  MoveL 4740 to (-40.39, 151.7, 78.65) mm, rotated rx -180 ry 0 rz 180 deg; joints [-52.89, -15.203, 87.582, 77.101, 54.898, -68.284]
  MoveL 4741 to (-40.39, 151.7, 78.65) mm, rotated rx -180 ry 0 rz 180 deg; joints [-52.89, -15.203, 87.582, 77.101, 54.898, -68.284]
  Call Extruder(10.98377)
  MoveL 4742 to (-40.44, 151.45, 78.65) mm, rotated rx 180 ry 0 rz -180 deg; joints [-52.871, -15.235, 87.606, 77.086, 54.882, -68.269]
  MoveL 4743 to (-40.44, 151.45, 78.65) mm, rotated rx 180 ry 0 rz -180 deg; joints [-52.871, -15.235, 87.606, 77.086, 54.882, -68.269]
  Call Extruder(11.11830)
  MoveL 4744 to (-40.49, 151.2, 78.65) mm, rotated rx 180 ry 0 rz 180 deg; joints [-52.853, -15.267, 87.629, 77.072, 54.867, -68.254]
  MoveL 4745 to (-40.49, 151.2, 78.65) mm, rotated rx 180 ry 0 rz 180 deg; joints [-52.853, -15.267, 87.629, 77.072, 54.867, -68.254]
  Call Extruder(11.25223)
  MoveL 4746 to (-40.54, 150.95, 78.65) mm, rotated rx 180 ry 0 rz 180 deg; joints [-52.834, -15.299, 87.653, 77.057, 54.851, -68.239]
  MoveL 4747 to (-40.54, 150.95, 78.65) mm, rotated rx 180 ry 0 rz 180 deg; joints [-52.834, -15.299, 87.653, 77.057, 54.851, -68.239]
  Call Extruder(11.40008)
  MoveL 4748 to (-40.59, 150.67, 78.65) mm, rotated rx 180 ry 0 rz 180 deg; joints [-52.812, -15.334, 87.679, 77.041, 54.833, -68.222]
  MoveL 4749 to (-40.59, 150.67, 78.65) mm, rotated rx 180 ry 0 rz 180 deg; joints [-52.812, -15.334, 87.679, 77.041, 54.833, -68.222]
  Call Extruder(11.56181)
  MoveL 4750 to (-40.64, 150.37, 78.65) mm, rotated rx -180 ry 0 rz -180 deg; joints [-52.787, -15.372, 87.707, 77.023, 54.812, -68.203]
  MoveL 4751 to (-40.64, 150.37, 78.65) mm, rotated rx -180 ry 0 rz -180 deg; joints [-52.787, -15.372, 87.707, 77.023, 54.812, -68.203]
  Call Extruder(11.72281)
  MoveL 4752 to (-40.69, 150.06, 78.65) mm, rotated rx -180 ry 0 rz 180 deg; joints [-52.762, -15.411, 87.735, 77.004, 54.791, -68.184]
  MoveL 4753 to (-40.69, 150.06, 78.65) mm, rotated rx -180 ry 0 rz 180 deg; joints [-52.762, -15.411, 87.735, 77.004, 54.791, -68.184]
  Call Extruder(11.88308)
  MoveL 4754 to (-40.74, 149.76, 78.65) mm, rotated rx 180 ry 0 rz 180 deg; joints [-52.737, -15.449, 87.762, 76.986, 54.771, -68.165]
  MoveL 4755 to (-40.74, 149.76, 78.65) mm, rotated rx 180 ry 0 rz 180 deg; joints [-52.737, -15.449, 87.762, 76.986, 54.771, -68.165]
  Call Extruder(12.04262)
  MoveL 4756 to (-40.78, 149.45, 78.65) mm, rotated rx 180 ry 0 rz 180 deg; joints [-52.712, -15.487, 87.79, 76.967, 54.75, -68.146]
  MoveL 4757 to (-40.78, 149.45, 78.65) mm, rotated rx 180 ry 0 rz 180 deg; joints [-52.712, -15.487, 87.79, 76.967, 54.75, -68.146]
  Call Extruder(12.20143)
  MoveL 4758 to (-40.83, 149.14, 78.65) mm, rotated rx -180 ry 0 rz -180 deg; joints [-52.687, -15.526, 87.818, 76.949, 54.729, -68.127]
  MoveL 4759 to (-40.83, 149.14, 78.65) mm, rotated rx -180 ry 0 rz -180 deg; joints [-52.687, -15.526, 87.818, 76.949, 54.729, -68.127]
  Call Extruder(12.38010)
  MoveL 4760 to (-40.88, 148.8, 78.65) mm, rotated rx 180 ry 0 rz 180 deg; joints [-52.658, -15.568, 87.849, 76.927, 54.704, -68.106]
  MoveL 4761 to (-40.88, 148.8, 78.65) mm, rotated rx 180 ry 0 rz 180 deg; joints [-52.658, -15.568, 87.849, 76.927, 54.704, -68.106]
  Call Extruder(12.57854)
  MoveL 4762 to (-40.92, 148.41, 78.65) mm, rotated rx 180 ry 0 rz 180 deg; joints [-52.624, -15.615, 87.883, 76.903, 54.675, -68.081]
  MoveL 4763 to (-40.92, 148.41, 78.65) mm, rotated rx 180 ry 0 rz 180 deg; joints [-52.624, -15.615, 87.883, 76.903, 54.675, -68.081]
  Call Extruder(12.77611)
  MoveL 4764 to (-40.97, 148.02, 78.65) mm, rotated rx 180 ry 0 rz -180 deg; joints [-52.59, -15.662, 87.917, 76.878, 54.647, -68.057]
  MoveL 4765 to (-40.97, 148.02, 78.65) mm, rotated rx 180 ry 0 rz -180 deg; joints [-52.59, -15.662, 87.917, 76.878, 54.647, -68.057]
  Call Extruder(12.97282)
  MoveL 4766 to (-41.02, 147.63, 78.65) mm, rotated rx -180 ry 0 rz 180 deg; joints [-52.556, -15.709, 87.951, 76.854, 54.618, -68.032]
  MoveL 4767 to (-41.02, 147.63, 78.65) mm, rotated rx -180 ry 0 rz 180 deg; joints [-52.556, -15.709, 87.951, 76.854, 54.618, -68.032]
  Call Extruder(13.16866)
  MoveL 4768 to (-41.06, 147.25, 78.65) mm, rotated rx 180 ry 0 rz 180 deg; joints [-52.521, -15.756, 87.985, 76.829, 54.589, -68.008]
  MoveL 4769 to (-41.06, 147.25, 78.65) mm, rotated rx 180 ry 0 rz 180 deg; joints [-52.521, -15.756, 87.985, 76.829, 54.589, -68.008]
  Call Extruder(13.46406)
  MoveL 4770 to (-41.11, 146.66, 78.65) mm, rotated rx -180 ry 0 rz 180 deg; joints [-52.466, -15.826, 88.036, 76.79, 54.543, -67.97]
  MoveL 4771 to (-41.11, 146.66, 78.65) mm, rotated rx -180 ry 0 rz 180 deg; joints [-52.466, -15.826, 88.036, 76.79, 54.543, -67.97]
  Call Extruder(13.75812)
  MoveL 4772 to (-41.15, 146.07, 78.65) mm, rotated rx 180 ry 0 rz 180 deg; joints [-52.411, -15.895, 88.086, 76.751, 54.496, -67.932]
  MoveL 4773 to (-41.15, 146.07, 78.65) mm, rotated rx 180 ry 0 rz 180 deg; joints [-52.411, -15.895, 88.086, 76.751, 54.496, -67.932]
  Call Extruder(14.05086)
  MoveL 4774 to (-41.2, 145.48, 78.65) mm, rotated rx -180 ry 0 rz 180 deg; joints [-52.355, -15.964, 88.136, 76.712, 54.449, -67.894]
  MoveL 4775 to (-41.2, 145.48, 78.65) mm, rotated rx -180 ry 0 rz 180 deg; joints [-52.355, -15.964, 88.136, 76.712, 54.449, -67.894]
  Call Extruder(14.62431)
  MoveL 4776 to (-41.25, 144.32, 78.65) mm, rotated rx -180 ry 0 rz 180 deg; joints [-52.239, -16.097, 88.231, 76.632, 54.349, -67.818]
  MoveL 4777 to (-41.25, 144.32, 78.65) mm, rotated rx -180 ry 0 rz 180 deg; joints [-52.239, -16.097, 88.231, 76.632, 54.349, -67.818]
  Call Extruder(15.33827)
  MoveL 4778 to (-41.29, 142.86, 78.65) mm, rotated rx 180 ry 0 rz 180 deg; joints [-52.09, -16.261, 88.348, 76.53, 54.222, -67.722]
  Call Extruder(57.40309)
  MoveL 4779 to (-41.29, 57.14, 78.65) mm, rotated rx 180 ry 0 rz 180 deg; joints [-40.759, -24.748, 93.754, 67.429, 44.994, -59.555]
  Call Extruder(57.83164)
  MoveL 4780 to (-41.27, 56.26, 78.65) mm, rotated rx 180 ry 0 rz 180 deg; joints [-40.614, -24.821, 93.795, 67.296, 44.882, -59.439]
  MoveL 4781 to (-41.27, 56.26, 78.65) mm, rotated rx 180 ry 0 rz 180 deg; joints [-40.614, -24.821, 93.795, 67.296, 44.882, -59.439]
  Call Extruder(58.40509)
  MoveL 4782 to (-41.22, 55.1, 78.65) mm, rotated rx -180 ry 0 rz 180 deg; joints [-40.419, -24.917, 93.848, 67.115, 44.73, -59.283]
  MoveL 4783 to (-41.22, 55.1, 78.65) mm, rotated rx -180 ry 0 rz 180 deg; joints [-40.419, -24.917, 93.848, 67.115, 44.73, -59.283]
  Call Extruder(58.83941)
  MoveL 4784 to (-41.18, 54.23, 78.65) mm, rotated rx 180 ry 0 rz 180 deg; joints [-40.269, -24.987, 93.887, 66.976, 44.613, -59.164]
  MoveL 4785 to (-41.18, 54.23, 78.65) mm, rotated rx 180 ry 0 rz 180 deg; joints [-40.269, -24.987, 93.887, 66.976, 44.613, -59.164]
  Call Extruder(59.13347)
  MoveL 4786 to (-41.13, 53.64, 78.65) mm, rotated rx 180 ry 0 rz -180 deg; joints [-40.165, -25.033, 93.912, 66.882, 44.532, -59.084]
  MoveL 4787 to (-41.13, 53.64, 78.65) mm, rotated rx 180 ry 0 rz -180 deg; joints [-40.165, -25.033, 93.912, 66.882, 44.532, -59.084]
  Call Extruder(59.42887)
  MoveL 4788 to (-41.09, 53.05, 78.65) mm, rotated rx -180 ry 0 rz 180 deg; joints [-40.062, -25.078, 93.937, 66.787, 44.452, -59.003]
  MoveL 4789 to (-41.09, 53.05, 78.65) mm, rotated rx -180 ry 0 rz 180 deg; joints [-40.062, -25.078, 93.937, 66.787, 44.452, -59.003]
  Call Extruder(59.67511)
  MoveL 4790 to (-41.04, 52.56, 78.65) mm, rotated rx -180 ry 0 rz 180 deg; joints [-39.975, -25.115, 93.958, 66.707, 44.384, -58.935]
  MoveL 4791 to (-41.04, 52.56, 78.65) mm, rotated rx -180 ry 0 rz 180 deg; joints [-39.975, -25.115, 93.958, 66.707, 44.384, -58.935]
  Call Extruder(59.87182)
  MoveL 4792 to (-40.99, 52.17, 78.65) mm, rotated rx 180 ry 0 rz 180 deg; joints [-39.904, -25.143, 93.973, 66.643, 44.328, -58.881]
  MoveL 4793 to (-40.99, 52.17, 78.65) mm, rotated rx 180 ry 0 rz 180 deg; joints [-39.904, -25.143, 93.973, 66.643, 44.328, -58.881]
  Call Extruder(60.06939)
  MoveL 4794 to (-40.95, 51.78, 78.65) mm, rotated rx -180 ry 0 rz -180 deg; joints [-39.833, -25.171, 93.989, 66.579, 44.273, -58.827]
  MoveL 4795 to (-40.95, 51.78, 78.65) mm, rotated rx -180 ry 0 rz -180 deg; joints [-39.833, -25.171, 93.989, 66.579, 44.273, -58.827]
  Call Extruder(60.26783)
  MoveL 4796 to (-40.9, 51.4, 78.65) mm, rotated rx 180 ry 0 rz 180 deg; joints [-39.763, -25.199, 94.004, 66.514, 44.217, -58.773]
  MoveL 4797 to (-40.9, 51.4, 78.65) mm, rotated rx 180 ry 0 rz 180 deg; joints [-39.763, -25.199, 94.004, 66.514, 44.217, -58.773]
  Call Extruder(60.46714)
  MoveL 4798 to (-40.86, 51.01, 78.65) mm, rotated rx 180 ry 0 rz 180 deg; joints [-39.692, -25.227, 94.02, 66.45, 44.162, -58.718]
  MoveL 4799 to (-40.86, 51.01, 78.65) mm, rotated rx 180 ry 0 rz 180 deg; joints [-39.692, -25.227, 94.02, 66.45, 44.162, -58.718]
  Call Extruder(60.62596)
  MoveL 4800 to (-40.81, 50.7, 78.65) mm, rotated rx 180 ry 0 rz 180 deg; joints [-39.634, -25.248, 94.031, 66.398, 44.116, -58.675]
  MoveL 4801 to (-40.81, 50.7, 78.65) mm, rotated rx 180 ry 0 rz 180 deg; joints [-39.634, -25.248, 94.031, 66.398, 44.116, -58.675]
  Call Extruder(60.78550)
  MoveL 4802 to (-40.76, 50.4, 78.65) mm, rotated rx 180 ry 0 rz 180 deg; joints [-39.576, -25.269, 94.043, 66.346, 44.07, -58.632]
  MoveL 4803 to (-40.76, 50.4, 78.65) mm, rotated rx 180 ry 0 rz 180 deg; joints [-39.576, -25.269, 94.043, 66.346, 44.07, -58.632]
  Call Extruder(60.94577)
  MoveL 4804 to (-40.71, 50.09, 78.65) mm, rotated rx -180 ry 0 rz 180 deg; joints [-39.518, -25.29, 94.054, 66.294, 44.025, -58.588]
  MoveL 4805 to (-40.71, 50.09, 78.65) mm, rotated rx -180 ry 0 rz 180 deg; joints [-39.518, -25.29, 94.054, 66.294, 44.025, -58.588]
  Call Extruder(61.10677)
  MoveL 4806 to (-40.66, 49.79, 78.65) mm, rotated rx -180 ry 0 rz 180 deg; joints [-39.46, -25.31, 94.065, 66.241, 43.979, -58.545]
  MoveL 4807 to (-40.66, 49.79, 78.65) mm, rotated rx -180 ry 0 rz 180 deg; joints [-39.46, -25.31, 94.065, 66.241, 43.979, -58.545]
  Call Extruder(61.26850)
  MoveL 4808 to (-40.61, 49.48, 78.65) mm, rotated rx 180 ry 0 rz 180 deg; joints [-39.402, -25.331, 94.077, 66.189, 43.933, -58.501]
  MoveL 4809 to (-40.61, 49.48, 78.65) mm, rotated rx 180 ry 0 rz 180 deg; joints [-39.402, -25.331, 94.077, 66.189, 43.933, -58.501]
  Call Extruder(61.43095)
  MoveL 4810 to (-40.57, 49.17, 78.65) mm, rotated rx 180 ry 0 rz 180 deg; joints [-39.344, -25.352, 94.088, 66.136, 43.888, -58.457]
  MoveL 4811 to (-40.57, 49.17, 78.65) mm, rotated rx 180 ry 0 rz 180 deg; joints [-39.344, -25.352, 94.088, 66.136, 43.888, -58.457]
  Call Extruder(61.56487)
  MoveL 4812 to (-40.52, 48.92, 78.65) mm, rotated rx -180 ry 0 rz 180 deg; joints [-39.296, -25.368, 94.096, 66.092, 43.849, -58.421]
  MoveL 4813 to (-40.52, 48.92, 78.65) mm, rotated rx -180 ry 0 rz 180 deg; joints [-39.296, -25.368, 94.096, 66.092, 43.849, -58.421]
  Call Extruder(61.69941)
  MoveL 4814 to (-40.47, 48.68, 78.65) mm, rotated rx 180 ry 0 rz 180 deg; joints [-39.247, -25.383, 94.105, 66.049, 43.81, -58.385]
  MoveL 4815 to (-40.47, 48.68, 78.65) mm, rotated rx 180 ry 0 rz 180 deg; joints [-39.247, -25.383, 94.105, 66.049, 43.81, -58.385]
  Call Extruder(61.83455)
  MoveL 4816 to (-40.42, 48.43, 78.65) mm, rotated rx 180 ry 0 rz 180 deg; joints [-39.198, -25.399, 94.114, 66.005, 43.772, -58.349]
  MoveL 4817 to (-40.42, 48.43, 78.65) mm, rotated rx 180 ry 0 rz 180 deg; joints [-39.198, -25.399, 94.114, 66.005, 43.772, -58.349]
  Call Extruder(61.97031)
  MoveL 4818 to (-40.37, 48.18, 78.65) mm, rotated rx 180 ry 0 rz 180 deg; joints [-39.149, -25.415, 94.122, 65.961, 43.733, -58.313]
  MoveL 4819 to (-40.37, 48.18, 78.65) mm, rotated rx 180 ry 0 rz 180 deg; joints [-39.149, -25.415, 94.122, 65.961, 43.733, -58.313]
  Call Extruder(62.10667)
  MoveL 4820 to (-40.32, 47.93, 78.65) mm, rotated rx -180 ry 0 rz 180 deg; joints [-39.1, -25.43, 94.131, 65.917, 43.694, -58.276]
  MoveL 4821 to (-40.32, 47.93, 78.65) mm, rotated rx -180 ry 0 rz 180 deg; joints [-39.1, -25.43, 94.131, 65.917, 43.694, -58.276]
  Call Extruder(62.24365)
  MoveL 4822 to (-40.27, 47.68, 78.65) mm, rotated rx 180 ry 0 rz 180 deg; joints [-39.051, -25.446, 94.139, 65.873, 43.656, -58.24]
  MoveL 4823 to (-40.27, 47.68, 78.65) mm, rotated rx 180 ry 0 rz 180 deg; joints [-39.051, -25.446, 94.139, 65.873, 43.656, -58.24]
  Call Extruder(62.38124)
  MoveL 4824 to (-40.22, 47.43, 78.65) mm, rotated rx -180 ry 0 rz 180 deg; joints [-39.002, -25.461, 94.148, 65.829, 43.617, -58.204]
  MoveL 4825 to (-40.22, 47.43, 78.65) mm, rotated rx -180 ry 0 rz 180 deg; joints [-39.002, -25.461, 94.148, 65.829, 43.617, -58.204]
  Call Extruder(62.49496)
  MoveL 4826 to (-40.17, 47.23, 78.65) mm, rotated rx 180 ry 0 rz 180 deg; joints [-38.962, -25.474, 94.154, 65.792, 43.585, -58.174]
  MoveL 4827 to (-40.17, 47.23, 78.65) mm, rotated rx 180 ry 0 rz 180 deg; joints [-38.962, -25.474, 94.154, 65.792, 43.585, -58.174]
  Call Extruder(62.60914)
  MoveL 4828 to (-40.13, 47.02, 78.65) mm, rotated rx -180 ry 0 rz 180 deg; joints [-38.921, -25.486, 94.161, 65.755, 43.552, -58.143]
  MoveL 4829 to (-40.13, 47.02, 78.65) mm, rotated rx -180 ry 0 rz 180 deg; joints [-38.921, -25.486, 94.161, 65.755, 43.552, -58.143]
  Call Extruder(62.72378)
  MoveL 4830 to (-40.08, 46.82, 78.65) mm, rotated rx -180 ry 0 rz 180 deg; joints [-38.88, -25.498, 94.168, 65.719, 43.52, -58.113]
  MoveL 4831 to (-40.08, 46.82, 78.65) mm, rotated rx -180 ry 0 rz 180 deg; joints [-38.88, -25.498, 94.168, 65.719, 43.52, -58.113]
  Call Extruder(62.83886)
  MoveL 4832 to (-40.04, 46.61, 78.65) mm, rotated rx 180 ry 0 rz 180 deg; joints [-38.839, -25.511, 94.175, 65.682, 43.488, -58.083]
  MoveL 4833 to (-40.04, 46.61, 78.65) mm, rotated rx 180 ry 0 rz 180 deg; joints [-38.839, -25.511, 94.175, 65.682, 43.488, -58.083]
  Call Extruder(62.96110)
  MoveL 4834 to (-39.98, 46.4, 78.65) mm, rotated rx 180 ry 0 rz -180 deg; joints [-38.795, -25.523, 94.181, 65.643, 43.452, -58.051]
  MoveL 4835 to (-39.98, 46.4, 78.65) mm, rotated rx 180 ry 0 rz -180 deg; joints [-38.795, -25.523, 94.181, 65.643, 43.452, -58.051]
  Call Extruder(63.09076)
  MoveL 4836 to (-39.92, 46.18, 78.65) mm, rotated rx 180 ry 0 rz 180 deg; joints [-38.748, -25.534, 94.187, 65.601, 43.414, -58.018]
  MoveL 4837 to (-39.92, 46.18, 78.65) mm, rotated rx 180 ry 0 rz 180 deg; joints [-38.748, -25.534, 94.187, 65.601, 43.414, -58.018]
  Call Extruder(63.22099)
  MoveL 4838 to (-39.85, 45.95, 78.65) mm, rotated rx -180 ry 0 rz 180 deg; joints [-38.7, -25.546, 94.193, 65.56, 43.376, -57.984]
  MoveL 4839 to (-39.85, 45.95, 78.65) mm, rotated rx -180 ry 0 rz 180 deg; joints [-38.7, -25.546, 94.193, 65.56, 43.376, -57.984]
  Call Extruder(63.35179)
  MoveL 4840 to (-39.78, 45.73, 78.65) mm, rotated rx -180 ry 0 rz 180 deg; joints [-38.653, -25.557, 94.2, 65.518, 43.338, -57.951]
  MoveL 4841 to (-39.78, 45.73, 78.65) mm, rotated rx -180 ry 0 rz 180 deg; joints [-38.653, -25.557, 94.2, 65.518, 43.338, -57.951]
  Call Extruder(63.48315)
  MoveL 4842 to (-39.71, 45.51, 78.65) mm, rotated rx 180 ry 0 rz 180 deg; joints [-38.605, -25.569, 94.206, 65.476, 43.3, -57.917]
  MoveL 4843 to (-39.71, 45.51, 78.65) mm, rotated rx 180 ry 0 rz 180 deg; joints [-38.605, -25.569, 94.206, 65.476, 43.3, -57.917]
  Call Extruder(63.59505)
  MoveL 4844 to (-39.65, 45.32, 78.65) mm, rotated rx 180 ry 0 rz 180 deg; joints [-38.565, -25.578, 94.211, 65.441, 43.268, -57.889]
  MoveL 4845 to (-39.65, 45.32, 78.65) mm, rotated rx 180 ry 0 rz 180 deg; joints [-38.565, -25.578, 94.211, 65.441, 43.268, -57.889]
  Call Extruder(63.70739)
  MoveL 4846 to (-39.59, 45.13, 78.65) mm, rotated rx 180 ry 0 rz 180 deg; joints [-38.524, -25.587, 94.216, 65.405, 43.235, -57.86]
  MoveL 4847 to (-39.59, 45.13, 78.65) mm, rotated rx 180 ry 0 rz 180 deg; joints [-38.524, -25.587, 94.216, 65.405, 43.235, -57.86]
  Call Extruder(63.82018)
  MoveL 4848 to (-39.53, 44.94, 78.65) mm, rotated rx 180 ry 0 rz 180 deg; joints [-38.483, -25.596, 94.221, 65.37, 43.202, -57.832]
  MoveL 4849 to (-39.53, 44.94, 78.65) mm, rotated rx 180 ry 0 rz 180 deg; joints [-38.483, -25.596, 94.221, 65.37, 43.202, -57.832]
  Call Extruder(63.93342)
  MoveL 4850 to (-39.47, 44.75, 78.65) mm, rotated rx 180 ry 0 rz 180 deg; joints [-38.443, -25.605, 94.226, 65.334, 43.169, -57.803]
  MoveL 4851 to (-39.47, 44.75, 78.65) mm, rotated rx 180 ry 0 rz 180 deg; joints [-38.443, -25.605, 94.226, 65.334, 43.169, -57.803]
  Call Extruder(64.04710)
  MoveL 4852 to (-39.41, 44.56, 78.65) mm, rotated rx 180 ry 0 rz 180 deg; joints [-38.402, -25.614, 94.231, 65.298, 43.137, -57.774]
  MoveL 4853 to (-39.41, 44.56, 78.65) mm, rotated rx 180 ry 0 rz 180 deg; joints [-38.402, -25.614, 94.231, 65.298, 43.137, -57.774]
  Call Extruder(64.22906)
  MoveL 4854 to (-39.29, 44.27, 78.65) mm, rotated rx 180 ry 0 rz 180 deg; joints [-38.335, -25.626, 94.237, 65.241, 43.083, -57.729]
  MoveL 4855 to (-39.29, 44.27, 78.65) mm, rotated rx 180 ry 0 rz 180 deg; joints [-38.335, -25.626, 94.237, 65.241, 43.083, -57.729]
  Call Extruder(64.41178)
  MoveL 4856 to (-39.17, 43.98, 78.65) mm, rotated rx -180 ry 0 rz -180 deg; joints [-38.269, -25.637, 94.243, 65.184, 43.028, -57.684]
  MoveL 4857 to (-39.17, 43.98, 78.65) mm, rotated rx -180 ry 0 rz -180 deg; joints [-38.269, -25.637, 94.243, 65.184, 43.028, -57.684]
  Call Extruder(64.58219)
  MoveL 4858 to (-39.05, 43.71, 78.65) mm, rotated rx 180 ry 0 rz 180 deg; joints [-38.207, -25.647, 94.249, 65.131, 42.978, -57.643]
  MoveL 4859 to (-39.05, 43.71, 78.65) mm, rotated rx 180 ry 0 rz 180 deg; joints [-38.207, -25.647, 94.249, 65.131, 42.978, -57.643]
  Call Extruder(64.74017)
  MoveL 4860 to (-38.94, 43.46, 78.65) mm, rotated rx -180 ry 0 rz -180 deg; joints [-38.149, -25.656, 94.253, 65.081, 42.931, -57.604]
  MoveL 4861 to (-38.94, 43.46, 78.65) mm, rotated rx -180 ry 0 rz -180 deg; joints [-38.149, -25.656, 94.253, 65.081, 42.931, -57.604]
  Call Extruder(64.89876)
  MoveL 4862 to (-38.84, 43.21, 78.65) mm, rotated rx 180 ry 0 rz 180 deg; joints [-38.092, -25.666, 94.258, 65.032, 42.884, -57.565]
  MoveL 4863 to (-38.84, 43.21, 78.65) mm, rotated rx 180 ry 0 rz 180 deg; joints [-38.092, -25.666, 94.258, 65.032, 42.884, -57.565]
  Call Extruder(65.10492)
  MoveL 4864 to (-38.66, 42.91, 78.65) mm, rotated rx 180 ry 0 rz 180 deg; joints [-38.016, -25.672, 94.262, 64.969, 42.821, -57.517]
  MoveL 4865 to (-38.66, 42.91, 78.65) mm, rotated rx 180 ry 0 rz 180 deg; joints [-38.016, -25.672, 94.262, 64.969, 42.821, -57.517]
  Call Extruder(65.31187)
  MoveL 4866 to (-38.49, 42.6, 78.65) mm, rotated rx 180 ry 0 rz 180 deg; joints [-37.939, -25.678, 94.265, 64.906, 42.758, -57.469]
  MoveL 4867 to (-38.49, 42.6, 78.65) mm, rotated rx 180 ry 0 rz 180 deg; joints [-37.939, -25.678, 94.265, 64.906, 42.758, -57.469]
  Call Extruder(65.51959)
  MoveL 4868 to (-38.31, 42.3, 78.65) mm, rotated rx 180 ry 0 rz 180 deg; joints [-37.863, -25.685, 94.269, 64.842, 42.695, -57.42]
  MoveL 4869 to (-38.31, 42.3, 78.65) mm, rotated rx 180 ry 0 rz 180 deg; joints [-37.863, -25.685, 94.269, 64.842, 42.695, -57.42]
  Call Extruder(65.72809)
  MoveL 4870 to (-38.14, 41.99, 78.65) mm, rotated rx 180 ry 0 rz -180 deg; joints [-37.787, -25.691, 94.272, 64.779, 42.632, -57.372]
  MoveL 4871 to (-38.14, 41.99, 78.65) mm, rotated rx 180 ry 0 rz -180 deg; joints [-37.787, -25.691, 94.272, 64.779, 42.632, -57.372]
  Call Extruder(65.90765)
  MoveL 4872 to (-37.96, 41.75, 78.65) mm, rotated rx -180 ry 0 rz 180 deg; joints [-37.72, -25.693, 94.273, 64.725, 42.577, -57.332]
  MoveL 4873 to (-37.96, 41.75, 78.65) mm, rotated rx -180 ry 0 rz 180 deg; joints [-37.72, -25.693, 94.273, 64.725, 42.577, -57.332]
  Call Extruder(66.24108)
  MoveL 4874 to (-37.63, 41.3, 78.65) mm, rotated rx 180 ry 0 rz 180 deg; joints [-37.598, -25.695, 94.274, 64.626, 42.474, -57.259]
  MoveL 4875 to (-37.63, 41.3, 78.65) mm, rotated rx 180 ry 0 rz 180 deg; joints [-37.598, -25.695, 94.274, 64.626, 42.474, -57.259]
  Call Extruder(66.57570)
  MoveL 4876 to (-37.3, 40.85, 78.65) mm, rotated rx 180 ry 0 rz 180 deg; joints [-37.475, -25.697, 94.275, 64.527, 42.371, -57.185]
  Call Extruder(67.40363)
  MoveL 4877 to (-36.39, 39.81, 78.65) mm, rotated rx 180 ry 0 rz 180 deg; joints [-37.173, -25.684, 94.268, 64.289, 42.115, -57.012]
  Call Extruder(68.23154)
  MoveL 4878 to (-35.35, 38.9, 78.65) mm, rotated rx -180 ry 0 rz 180 deg; joints [-36.876, -25.647, 94.249, 64.063, 41.859, -56.855]
  Call Extruder(68.39885)
  MoveL 4879 to (-35.13, 38.73, 78.65) mm, rotated rx -180 ry 0 rz 180 deg; joints [-36.818, -25.636, 94.243, 64.02, 41.808, -56.826]
  MoveL 4880 to (-35.13, 38.73, 78.65) mm, rotated rx -180 ry 0 rz 180 deg; joints [-36.818, -25.636, 94.243, 64.02, 41.808, -56.826]
  Call Extruder(68.73227)
  MoveL 4881 to (-34.68, 38.41, 78.65) mm, rotated rx 180 ry 0 rz -180 deg; joints [-36.701, -25.615, 94.231, 63.934, 41.706, -56.767]
  MoveL 4882 to (-34.68, 38.41, 78.65) mm, rotated rx 180 ry 0 rz -180 deg; joints [-36.701, -25.615, 94.231, 63.934, 41.706, -56.767]
  Call Extruder(69.06451)
  MoveL 4883 to (-34.22, 38.08, 78.65) mm, rotated rx 180 ry 0 rz 180 deg; joints [-36.584, -25.593, 94.219, 63.848, 41.603, -56.709]
  MoveL 4884 to (-34.22, 38.08, 78.65) mm, rotated rx 180 ry 0 rz 180 deg; joints [-36.584, -25.593, 94.219, 63.848, 41.603, -56.709]
  Call Extruder(69.18222)
  MoveL 4885 to (-34.05, 37.98, 78.65) mm, rotated rx 180 ry 0 rz -180 deg; joints [-36.544, -25.582, 94.213, 63.82, 41.568, -56.691]
  MoveL 4886 to (-34.05, 37.98, 78.65) mm, rotated rx 180 ry 0 rz -180 deg; joints [-36.544, -25.582, 94.213, 63.82, 41.568, -56.691]
  Call Extruder(69.38994)
  MoveL 4887 to (-33.75, 37.8, 78.65) mm, rotated rx 180 ry 0 rz 180 deg; joints [-36.474, -25.564, 94.203, 63.77, 41.506, -56.658]
  MoveL 4888 to (-33.75, 37.8, 78.65) mm, rotated rx 180 ry 0 rz 180 deg; joints [-36.474, -25.564, 94.203, 63.77, 41.506, -56.658]
  Call Extruder(69.59688)
  MoveL 4889 to (-33.45, 37.63, 78.65) mm, rotated rx -180 ry 0 rz 180 deg; joints [-36.403, -25.546, 94.193, 63.72, 41.443, -56.626]
  MoveL 4890 to (-33.45, 37.63, 78.65) mm, rotated rx -180 ry 0 rz 180 deg; joints [-36.403, -25.546, 94.193, 63.72, 41.443, -56.626]
  Call Extruder(69.80304)
  MoveL 4891 to (-33.14, 37.45, 78.65) mm, rotated rx 180 ry 0 rz -180 deg; joints [-36.333, -25.527, 94.183, 63.67, 41.381, -56.594]
  MoveL 4892 to (-33.14, 37.45, 78.65) mm, rotated rx 180 ry 0 rz -180 deg; joints [-36.333, -25.527, 94.183, 63.67, 41.381, -56.594]
  Call Extruder(69.98473)
  MoveL 4893 to (-32.86, 37.31, 78.65) mm, rotated rx 180 ry 0 rz 180 deg; joints [-36.272, -25.509, 94.173, 63.628, 41.326, -56.567]
  MoveL 4894 to (-32.86, 37.31, 78.65) mm, rotated rx 180 ry 0 rz 180 deg; joints [-36.272, -25.509, 94.173, 63.628, 41.326, -56.567]
  Call Extruder(70.14273)
  MoveL 4895 to (-32.62, 37.2, 78.65) mm, rotated rx 180 ry 0 rz 180 deg; joints [-36.221, -25.491, 94.164, 63.594, 41.28, -56.546]
  MoveL 4896 to (-32.62, 37.2, 78.65) mm, rotated rx 180 ry 0 rz 180 deg; joints [-36.221, -25.491, 94.164, 63.594, 41.28, -56.546]
  Call Extruder(70.30013)
  MoveL 4897 to (-32.37, 37.1, 78.65) mm, rotated rx 180 ry 0 rz -180 deg; joints [-36.17, -25.472, 94.154, 63.56, 41.234, -56.525]
  MoveL 4898 to (-32.37, 37.1, 78.65) mm, rotated rx 180 ry 0 rz -180 deg; joints [-36.17, -25.472, 94.154, 63.56, 41.234, -56.525]
  Call Extruder(70.48284)
  MoveL 4899 to (-32.08, 36.97, 78.65) mm, rotated rx 180 ry 0 rz 180 deg; joints [-36.112, -25.451, 94.142, 63.521, 41.18, -56.502]
  MoveL 4900 to (-32.08, 36.97, 78.65) mm, rotated rx 180 ry 0 rz 180 deg; joints [-36.112, -25.451, 94.142, 63.521, 41.18, -56.502]
  Call Extruder(70.66479)
  MoveL 4901 to (-31.78, 36.85, 78.65) mm, rotated rx 180 ry 0 rz 180 deg; joints [-36.053, -25.429, 94.13, 63.482, 41.127, -56.478]
  MoveL 4902 to (-31.78, 36.85, 78.65) mm, rotated rx 180 ry 0 rz 180 deg; joints [-36.053, -25.429, 94.13, 63.482, 41.127, -56.478]
  Call Extruder(70.81212)
  MoveL 4903 to (-31.54, 36.76, 78.65) mm, rotated rx 180 ry 0 rz 180 deg; joints [-36.006, -25.41, 94.12, 63.451, 41.084, -56.46]
  MoveL 4904 to (-31.54, 36.76, 78.65) mm, rotated rx 180 ry 0 rz 180 deg; joints [-36.006, -25.41, 94.12, 63.451, 41.084, -56.46]
  Call Extruder(70.92535)
  MoveL 4905 to (-31.35, 36.7, 78.65) mm, rotated rx 180 ry 0 rz 180 deg; joints [-35.971, -25.395, 94.111, 63.429, 41.052, -56.447]
  MoveL 4906 to (-31.35, 36.7, 78.65) mm, rotated rx 180 ry 0 rz 180 deg; joints [-35.971, -25.395, 94.111, 63.429, 41.052, -56.447]
  Call Extruder(71.03815)
  MoveL 4907 to (-31.17, 36.64, 78.65) mm, rotated rx -180 ry 0 rz 180 deg; joints [-35.936, -25.38, 94.103, 63.407, 41.02, -56.435]
  MoveL 4908 to (-31.17, 36.64, 78.65) mm, rotated rx -180 ry 0 rz 180 deg; joints [-35.936, -25.38, 94.103, 63.407, 41.02, -56.435]
  Call Extruder(71.15049)
  MoveL 4909 to (-30.98, 36.58, 78.65) mm, rotated rx -180 ry 0 rz -180 deg; joints [-35.901, -25.364, 94.095, 63.384, 40.988, -56.422]
  MoveL 4910 to (-30.98, 36.58, 78.65) mm, rotated rx -180 ry 0 rz -180 deg; joints [-35.901, -25.364, 94.095, 63.384, 40.988, -56.422]
  Call Extruder(71.26240)
  MoveL 4911 to (-30.79, 36.52, 78.65) mm, rotated rx 180 ry 0 rz 180 deg; joints [-35.867, -25.349, 94.086, 63.362, 40.956, -56.409]
  MoveL 4912 to (-30.79, 36.52, 78.65) mm, rotated rx 180 ry 0 rz 180 deg; joints [-35.867, -25.349, 94.086, 63.362, 40.956, -56.409]
  Call Extruder(71.38380)
  MoveL 4913 to (-30.58, 36.45, 78.65) mm, rotated rx -180 ry 0 rz 180 deg; joints [-35.829, -25.332, 94.077, 63.338, 40.921, -56.396]
  MoveL 4914 to (-30.58, 36.45, 78.65) mm, rotated rx -180 ry 0 rz 180 deg; joints [-35.829, -25.332, 94.077, 63.338, 40.921, -56.396]
  Call Extruder(71.51459)
  MoveL 4915 to (-30.36, 36.39, 78.65) mm, rotated rx 180 ry 0 rz 180 deg; joints [-35.788, -25.313, 94.067, 63.313, 40.883, -56.382]
  MoveL 4916 to (-30.36, 36.39, 78.65) mm, rotated rx 180 ry 0 rz 180 deg; joints [-35.788, -25.313, 94.067, 63.313, 40.883, -56.382]
  Call Extruder(71.64481)
  MoveL 4917 to (-30.14, 36.32, 78.65) mm, rotated rx 180 ry 0 rz 180 deg; joints [-35.748, -25.294, 94.056, 63.288, 40.846, -56.368]
  MoveL 4918 to (-30.14, 36.32, 78.65) mm, rotated rx 180 ry 0 rz 180 deg; joints [-35.748, -25.294, 94.056, 63.288, 40.846, -56.368]
  Call Extruder(71.77447)
  MoveL 4919 to (-29.91, 36.25, 78.65) mm, rotated rx 180 ry 0 rz 180 deg; joints [-35.708, -25.276, 94.046, 63.262, 40.809, -56.353]
  MoveL 4920 to (-29.91, 36.25, 78.65) mm, rotated rx 180 ry 0 rz 180 deg; joints [-35.708, -25.276, 94.046, 63.262, 40.809, -56.353]
  Call Extruder(71.90357)
  MoveL 4921 to (-29.69, 36.18, 78.65) mm, rotated rx 180 ry 0 rz 180 deg; joints [-35.668, -25.257, 94.036, 63.237, 40.771, -56.339]
  MoveL 4922 to (-29.69, 36.18, 78.65) mm, rotated rx 180 ry 0 rz 180 deg; joints [-35.668, -25.257, 94.036, 63.237, 40.771, -56.339]
  Call Extruder(72.01864)
  MoveL 4923 to (-29.48, 36.14, 78.65) mm, rotated rx 180 ry 0 rz 180 deg; joints [-35.634, -25.238, 94.026, 63.217, 40.74, -56.329]
  MoveL 4924 to (-29.48, 36.14, 78.65) mm, rotated rx 180 ry 0 rz 180 deg; joints [-35.634, -25.238, 94.026, 63.217, 40.74, -56.329]
  Call Extruder(72.13326)
  MoveL 4925 to (-29.28, 36.09, 78.65) mm, rotated rx 180 ry 0 rz 180 deg; joints [-35.601, -25.22, 94.016, 63.197, 40.708, -56.318]
  MoveL 4926 to (-29.28, 36.09, 78.65) mm, rotated rx 180 ry 0 rz 180 deg; joints [-35.601, -25.22, 94.016, 63.197, 40.708, -56.318]
  Call Extruder(72.24743)
  MoveL 4927 to (-29.08, 36.05, 78.65) mm, rotated rx 180 ry 0 rz 180 deg; joints [-35.567, -25.201, 94.005, 63.177, 40.676, -56.308]
  MoveL 4928 to (-29.08, 36.05, 78.65) mm, rotated rx 180 ry 0 rz 180 deg; joints [-35.567, -25.201, 94.005, 63.177, 40.676, -56.308]
  Call Extruder(72.36115)
  MoveL 4929 to (-28.87, 36, 78.65) mm, rotated rx 180 ry 0 rz 180 deg; joints [-35.533, -25.183, 93.995, 63.157, 40.644, -56.298]
  MoveL 4930 to (-28.87, 36, 78.65) mm, rotated rx 180 ry 0 rz 180 deg; joints [-35.533, -25.183, 93.995, 63.157, 40.644, -56.298]
  Call Extruder(72.48657)
  MoveL 4931 to (-28.65, 35.96, 78.65) mm, rotated rx 180 ry 0 rz 180 deg; joints [-35.497, -25.162, 93.984, 63.136, 40.61, -56.287]
  MoveL 4932 to (-28.65, 35.96, 78.65) mm, rotated rx 180 ry 0 rz 180 deg; joints [-35.497, -25.162, 93.984, 63.136, 40.61, -56.287]
  Call Extruder(72.62355)
  MoveL 4933 to (-28.4, 35.91, 78.65) mm, rotated rx 180 ry 0 rz 180 deg; joints [-35.457, -25.139, 93.971, 63.112, 40.572, -56.275]
  MoveL 4934 to (-28.4, 35.91, 78.65) mm, rotated rx 180 ry 0 rz 180 deg; joints [-35.457, -25.139, 93.971, 63.112, 40.572, -56.275]
  Call Extruder(72.75991)
  MoveL 4935 to (-28.15, 35.86, 78.65) mm, rotated rx -180 ry 0 rz 180 deg; joints [-35.417, -25.116, 93.959, 63.089, 40.534, -56.264]
  MoveL 4936 to (-28.15, 35.86, 78.65) mm, rotated rx -180 ry 0 rz 180 deg; joints [-35.417, -25.116, 93.959, 63.089, 40.534, -56.264]
  Call Extruder(72.89567)
  MoveL 4937 to (-27.9, 35.81, 78.65) mm, rotated rx 180 ry 0 rz 180 deg; joints [-35.377, -25.093, 93.946, 63.066, 40.496, -56.252]
  MoveL 4938 to (-27.9, 35.81, 78.65) mm, rotated rx 180 ry 0 rz 180 deg; joints [-35.377, -25.093, 93.946, 63.066, 40.496, -56.252]
  Call Extruder(73.03082)
  MoveL 4939 to (-27.65, 35.76, 78.65) mm, rotated rx -180 ry 0 rz 180 deg; joints [-35.337, -25.07, 93.933, 63.042, 40.458, -56.24]
  MoveL 4940 to (-27.65, 35.76, 78.65) mm, rotated rx -180 ry 0 rz 180 deg; joints [-35.337, -25.07, 93.933, 63.042, 40.458, -56.24]
  Call Extruder(73.16535)
  MoveL 4941 to (-27.4, 35.71, 78.65) mm, rotated rx 180 ry 0 rz -180 deg; joints [-35.297, -25.047, 93.92, 63.019, 40.42, -56.228]
  MoveL 4942 to (-27.4, 35.71, 78.65) mm, rotated rx 180 ry 0 rz -180 deg; joints [-35.297, -25.047, 93.92, 63.019, 40.42, -56.228]
  Call Extruder(73.29928)
  MoveL 4943 to (-27.15, 35.66, 78.65) mm, rotated rx -180 ry 0 rz 180 deg; joints [-35.258, -25.024, 93.908, 62.996, 40.383, -56.217]
  MoveL 4944 to (-27.15, 35.66, 78.65) mm, rotated rx -180 ry 0 rz 180 deg; joints [-35.258, -25.024, 93.908, 62.996, 40.383, -56.217]
  Call Extruder(73.44714)
  MoveL 4945 to (-26.87, 35.61, 78.65) mm, rotated rx -180 ry 0 rz 180 deg; joints [-35.215, -24.998, 93.893, 62.971, 40.342, -56.204]
  MoveL 4946 to (-26.87, 35.61, 78.65) mm, rotated rx -180 ry 0 rz 180 deg; joints [-35.215, -24.998, 93.893, 62.971, 40.342, -56.204]
  Call Extruder(73.60887)
  MoveL 4947 to (-26.57, 35.56, 78.65) mm, rotated rx -180 ry 0 rz 180 deg; joints [-35.168, -24.968, 93.877, 62.945, 40.297, -56.192]
  MoveL 4948 to (-26.57, 35.56, 78.65) mm, rotated rx -180 ry 0 rz 180 deg; joints [-35.168, -24.968, 93.877, 62.945, 40.297, -56.192]
  Call Extruder(73.76988)
  MoveL 4949 to (-26.26, 35.51, 78.65) mm, rotated rx 180 ry 0 rz 180 deg; joints [-35.122, -24.939, 93.861, 62.919, 40.253, -56.18]
  MoveL 4950 to (-26.26, 35.51, 78.65) mm, rotated rx 180 ry 0 rz 180 deg; joints [-35.122, -24.939, 93.861, 62.919, 40.253, -56.18]
  Call Extruder(73.93016)
  MoveL 4951 to (-25.96, 35.47, 78.65) mm, rotated rx 180 ry 0 rz -180 deg; joints [-35.075, -24.91, 93.844, 62.893, 40.208, -56.167]
  MoveL 4952 to (-25.96, 35.47, 78.65) mm, rotated rx 180 ry 0 rz -180 deg; joints [-35.075, -24.91, 93.844, 62.893, 40.208, -56.167]
  Call Extruder(74.08971)
  MoveL 4953 to (-25.65, 35.42, 78.65) mm, rotated rx -180 ry 0 rz 180 deg; joints [-35.029, -24.88, 93.828, 62.867, 40.164, -56.155]
  MoveL 4954 to (-25.65, 35.42, 78.65) mm, rotated rx -180 ry 0 rz 180 deg; joints [-35.029, -24.88, 93.828, 62.867, 40.164, -56.155]
  Call Extruder(74.24853)
  MoveL 4955 to (-25.34, 35.37, 78.65) mm, rotated rx -180 ry 0 rz 180 deg; joints [-34.983, -24.851, 93.812, 62.84, 40.12, -56.142]
  MoveL 4956 to (-25.34, 35.37, 78.65) mm, rotated rx -180 ry 0 rz 180 deg; joints [-34.983, -24.851, 93.812, 62.84, 40.12, -56.142]
  Call Extruder(74.42720)
  MoveL 4957 to (-25, 35.32, 78.65) mm, rotated rx 180 ry 0 rz 180 deg; joints [-34.932, -24.817, 93.793, 62.812, 40.071, -56.13]
  MoveL 4958 to (-25, 35.32, 78.65) mm, rotated rx 180 ry 0 rz 180 deg; joints [-34.932, -24.817, 93.793, 62.812, 40.071, -56.13]
  Call Extruder(74.62564)
  MoveL 4959 to (-24.61, 35.27, 78.65) mm, rotated rx 180 ry 0 rz 180 deg; joints [-34.877, -24.778, 93.771, 62.782, 40.017, -56.116]
  MoveL 4960 to (-24.61, 35.27, 78.65) mm, rotated rx 180 ry 0 rz 180 deg; joints [-34.877, -24.778, 93.771, 62.782, 40.017, -56.116]
  Call Extruder(74.82322)
  MoveL 4961 to (-24.22, 35.23, 78.65) mm, rotated rx 180 ry 0 rz 180 deg; joints [-34.821, -24.74, 93.75, 62.752, 39.963, -56.103]
  MoveL 4962 to (-24.22, 35.23, 78.65) mm, rotated rx 180 ry 0 rz 180 deg; joints [-34.821, -24.74, 93.75, 62.752, 39.963, -56.103]
  Call Extruder(75.01993)
  MoveL 4963 to (-23.83, 35.18, 78.65) mm, rotated rx 180 ry 0 rz -180 deg; joints [-34.766, -24.701, 93.728, 62.722, 39.909, -56.09]
  MoveL 4964 to (-23.83, 35.18, 78.65) mm, rotated rx 180 ry 0 rz -180 deg; joints [-34.766, -24.701, 93.728, 62.722, 39.909, -56.09]
  Call Extruder(75.21577)
  MoveL 4965 to (-23.45, 35.14, 78.65) mm, rotated rx 180 ry 0 rz 180 deg; joints [-34.711, -24.662, 93.706, 62.693, 39.856, -56.077]
  MoveL 4966 to (-23.45, 35.14, 78.65) mm, rotated rx 180 ry 0 rz 180 deg; joints [-34.711, -24.662, 93.706, 62.693, 39.856, -56.077]
  Call Extruder(75.51116)
  MoveL 4967 to (-22.86, 35.09, 78.65) mm, rotated rx -180 ry 0 rz 180 deg; joints [-34.631, -24.601, 93.672, 62.652, 39.777, -56.061]
  MoveL 4968 to (-22.86, 35.09, 78.65) mm, rotated rx -180 ry 0 rz 180 deg; joints [-34.631, -24.601, 93.672, 62.652, 39.777, -56.061]
  Call Extruder(75.80522)
  MoveL 4969 to (-22.27, 35.04, 78.65) mm, rotated rx -180 ry 0 rz 180 deg; joints [-34.552, -24.541, 93.638, 62.611, 39.699, -56.044]
  MoveL 4970 to (-22.27, 35.04, 78.65) mm, rotated rx -180 ry 0 rz 180 deg; joints [-34.552, -24.541, 93.638, 62.611, 39.699, -56.044]
  Call Extruder(76.09795)
  MoveL 4971 to (-21.68, 35, 78.65) mm, rotated rx 180 ry 0 rz 180 deg; joints [-34.473, -24.48, 93.604, 62.57, 39.621, -56.028]
  MoveL 4972 to (-21.68, 35, 78.65) mm, rotated rx 180 ry 0 rz 180 deg; joints [-34.473, -24.48, 93.604, 62.57, 39.621, -56.028]
  Call Extruder(76.67140)
  MoveL 4973 to (-20.52, 34.95, 78.65) mm, rotated rx 180 ry 0 rz 180 deg; joints [-34.326, -24.356, 93.534, 62.499, 39.475, -56.004]
  MoveL 4974 to (-20.52, 34.95, 78.65) mm, rotated rx 180 ry 0 rz 180 deg; joints [-34.326, -24.356, 93.534, 62.499, 39.475, -56.004]
  Call Extruder(77.38537)
  MoveL 4975 to (-19.06, 34.91, 78.65) mm, rotated rx 180 ry 0 rz 180 deg; joints [-34.146, -24.199, 93.445, 62.414, 39.294, -55.976]
  Call Extruder(194.23211)
  MoveL 4976 to (219.06, 34.91, 78.65) mm, rotated rx 180 ry 0 rz 180 deg; joints [-18.248, 7.691, 66.193, 49.907, 24.163, -47.302]
  Call Extruder(194.66067)
  MoveL 4977 to (219.94, 34.93, 78.65) mm, rotated rx -180 ry 0 rz 180 deg; joints [-18.218, 7.834, 66.031, 49.824, 24.153, -47.22]
  MoveL 4978 to (219.94, 34.93, 78.65) mm, rotated rx -180 ry 0 rz 180 deg; joints [-18.218, 7.834, 66.031, 49.824, 24.153, -47.22]
  Call Extruder(195.23412)
  MoveL 4979 to (221.1, 34.97, 78.65) mm, rotated rx -180 ry 0 rz 180 deg; joints [-18.181, 8.026, 65.813, 49.716, 24.143, -47.114]
  MoveL 4980 to (221.1, 34.97, 78.65) mm, rotated rx -180 ry 0 rz 180 deg; joints [-18.181, 8.026, 65.813, 49.716, 24.143, -47.114]
  Call Extruder(195.66843)
  MoveL 4981 to (221.97, 35.02, 78.65) mm, rotated rx 180 ry 0 rz -180 deg; joints [-18.154, 8.171, 65.646, 49.637, 24.136, -47.034]
  MoveL 4982 to (221.97, 35.02, 78.65) mm, rotated rx 180 ry 0 rz -180 deg; joints [-18.154, 8.171, 65.646, 49.637, 24.136, -47.034]
  Call Extruder(195.96249)
  MoveL 4983 to (222.56, 35.07, 78.65) mm, rotated rx -180 ry 0 rz -180 deg; joints [-18.138, 8.27, 65.533, 49.586, 24.134, -46.983]
  MoveL 4984 to (222.56, 35.07, 78.65) mm, rotated rx -180 ry 0 rz -180 deg; joints [-18.138, 8.27, 65.533, 49.586, 24.134, -46.983]
  Call Extruder(196.25788)
  MoveL 4985 to (223.15, 35.11, 78.65) mm, rotated rx 180 ry 0 rz -180 deg; joints [-18.121, 8.369, 65.42, 49.534, 24.131, -46.932]
  MoveL 4986 to (223.15, 35.11, 78.65) mm, rotated rx 180 ry 0 rz -180 deg; joints [-18.121, 8.369, 65.42, 49.534, 24.131, -46.932]
  Call Extruder(196.50411)
  MoveL 4987 to (223.64, 35.16, 78.65) mm, rotated rx 180 ry 0 rz 180 deg; joints [-18.109, 8.452, 65.325, 49.492, 24.13, -46.89]
  MoveL 4988 to (223.64, 35.16, 78.65) mm, rotated rx 180 ry 0 rz 180 deg; joints [-18.109, 8.452, 65.325, 49.492, 24.13, -46.89]
  Call Extruder(196.70082)
  MoveL 4989 to (224.03, 35.21, 78.65) mm, rotated rx -180 ry 0 rz -180 deg; joints [-18.1, 8.518, 65.249, 49.461, 24.13, -46.858]
  MoveL 4990 to (224.03, 35.21, 78.65) mm, rotated rx -180 ry 0 rz -180 deg; joints [-18.1, 8.518, 65.249, 49.461, 24.13, -46.858]
  Call Extruder(196.89839)
  MoveL 4991 to (224.42, 35.25, 78.65) mm, rotated rx 180 ry 0 rz 180 deg; joints [-18.091, 8.584, 65.173, 49.429, 24.13, -46.826]
  MoveL 4992 to (224.42, 35.25, 78.65) mm, rotated rx 180 ry 0 rz 180 deg; joints [-18.091, 8.584, 65.173, 49.429, 24.13, -46.826]
  Call Extruder(197.09684)
  MoveL 4993 to (224.8, 35.3, 78.65) mm, rotated rx 180 ry 0 rz 180 deg; joints [-18.082, 8.65, 65.097, 49.397, 24.13, -46.794]
  MoveL 4994 to (224.8, 35.3, 78.65) mm, rotated rx 180 ry 0 rz 180 deg; joints [-18.082, 8.65, 65.097, 49.397, 24.13, -46.794]
  Call Extruder(197.29615)
  MoveL 4995 to (225.19, 35.34, 78.65) mm, rotated rx 180 ry 0 rz 180 deg; joints [-18.073, 8.717, 65.02, 49.365, 24.13, -46.762]
  MoveL 4996 to (225.19, 35.34, 78.65) mm, rotated rx 180 ry 0 rz 180 deg; joints [-18.073, 8.717, 65.02, 49.365, 24.13, -46.762]
  Call Extruder(197.45497)
  MoveL 4997 to (225.5, 35.39, 78.65) mm, rotated rx -180 ry 0 rz 180 deg; joints [-18.068, 8.77, 64.959, 49.342, 24.131, -46.738]
  MoveL 4998 to (225.5, 35.39, 78.65) mm, rotated rx -180 ry 0 rz 180 deg; joints [-18.068, 8.77, 64.959, 49.342, 24.131, -46.738]
  Call Extruder(197.61451)
  MoveL 4999 to (225.8, 35.44, 78.65) mm, rotated rx -180 ry 0 rz 180 deg; joints [-18.062, 8.823, 64.898, 49.319, 24.132, -46.714]
  MoveL 5000 to (225.8, 35.44, 78.65) mm, rotated rx -180 ry 0 rz 180 deg; joints [-18.062, 8.823, 64.898, 49.319, 24.132, -46.714]
  Call Extruder(197.77479)
  MoveL 5001 to (226.11, 35.49, 78.65) mm, rotated rx 180 ry 0 rz -180 deg; joints [-18.056, 8.876, 64.837, 49.296, 24.133, -46.691]
  MoveL 5002 to (226.11, 35.49, 78.65) mm, rotated rx 180 ry 0 rz -180 deg; joints [-18.056, 8.876, 64.837, 49.296, 24.133, -46.691]
  Call Extruder(197.93579)
  MoveL 5003 to (226.41, 35.54, 78.65) mm, rotated rx -180 ry 0 rz 180 deg; joints [-18.051, 8.929, 64.775, 49.272, 24.135, -46.667]
  MoveL 5004 to (226.41, 35.54, 78.65) mm, rotated rx -180 ry 0 rz 180 deg; joints [-18.051, 8.929, 64.775, 49.272, 24.135, -46.667]
  Call Extruder(198.09752)
  MoveL 5005 to (226.72, 35.59, 78.65) mm, rotated rx 180 ry 0 rz 180 deg; joints [-18.045, 8.982, 64.714, 49.249, 24.136, -46.643]
  MoveL 5006 to (226.72, 35.59, 78.65) mm, rotated rx 180 ry 0 rz 180 deg; joints [-18.045, 8.982, 64.714, 49.249, 24.136, -46.643]
  Call Extruder(198.25998)
  MoveL 5007 to (227.02, 35.64, 78.65) mm, rotated rx 180 ry 0 rz 180 deg; joints [-18.039, 9.035, 64.652, 49.225, 24.137, -46.619]
  MoveL 5008 to (227.02, 35.64, 78.65) mm, rotated rx 180 ry 0 rz 180 deg; joints [-18.039, 9.035, 64.652, 49.225, 24.137, -46.619]
  Call Extruder(198.39391)
  MoveL 5009 to (227.27, 35.68, 78.65) mm, rotated rx 180 ry 0 rz -180 deg; joints [-18.036, 9.08, 64.601, 49.207, 24.139, -46.6]
  MoveL 5010 to (227.27, 35.68, 78.65) mm, rotated rx 180 ry 0 rz -180 deg; joints [-18.036, 9.08, 64.601, 49.207, 24.139, -46.6]
  Call Extruder(198.52845)
  MoveL 5011 to (227.52, 35.73, 78.65) mm, rotated rx -180 ry 0 rz 180 deg; joints [-18.033, 9.123, 64.55, 49.19, 24.141, -46.582]
  MoveL 5012 to (227.52, 35.73, 78.65) mm, rotated rx -180 ry 0 rz 180 deg; joints [-18.033, 9.123, 64.55, 49.19, 24.141, -46.582]
  Call Extruder(198.66359)
  MoveL 5013 to (227.77, 35.78, 78.65) mm, rotated rx 180 ry 0 rz 180 deg; joints [-18.029, 9.167, 64.499, 49.172, 24.144, -46.564]
  MoveL 5014 to (227.77, 35.78, 78.65) mm, rotated rx 180 ry 0 rz 180 deg; joints [-18.029, 9.167, 64.499, 49.172, 24.144, -46.564]
  Call Extruder(198.79935)
  MoveL 5015 to (228.02, 35.83, 78.65) mm, rotated rx 180 ry 0 rz 180 deg; joints [-18.026, 9.211, 64.448, 49.154, 24.146, -46.545]
  MoveL 5016 to (228.02, 35.83, 78.65) mm, rotated rx 180 ry 0 rz 180 deg; joints [-18.026, 9.211, 64.448, 49.154, 24.146, -46.545]
  Call Extruder(198.93572)
  MoveL 5017 to (228.27, 35.88, 78.65) mm, rotated rx 180 ry 0 rz -180 deg; joints [-18.022, 9.256, 64.397, 49.137, 24.148, -46.527]
  MoveL 5018 to (228.27, 35.88, 78.65) mm, rotated rx 180 ry 0 rz -180 deg; joints [-18.022, 9.256, 64.397, 49.137, 24.148, -46.527]
  Call Extruder(199.07270)
  MoveL 5019 to (228.52, 35.93, 78.65) mm, rotated rx 180 ry 0 rz 180 deg; joints [-18.019, 9.3, 64.346, 49.119, 24.15, -46.508]
  MoveL 5020 to (228.52, 35.93, 78.65) mm, rotated rx 180 ry 0 rz 180 deg; joints [-18.019, 9.3, 64.346, 49.119, 24.15, -46.508]
  Call Extruder(199.21029)
  MoveL 5021 to (228.77, 35.98, 78.65) mm, rotated rx 180 ry 0 rz 180 deg; joints [-18.015, 9.344, 64.295, 49.101, 24.152, -46.49]
  MoveL 5022 to (228.77, 35.98, 78.65) mm, rotated rx 180 ry 0 rz 180 deg; joints [-18.015, 9.344, 64.295, 49.101, 24.152, -46.49]
  Call Extruder(199.32400)
  MoveL 5023 to (228.97, 36.03, 78.65) mm, rotated rx 180 ry 0 rz 180 deg; joints [-18.013, 9.38, 64.252, 49.087, 24.154, -46.475]
  MoveL 5024 to (228.97, 36.03, 78.65) mm, rotated rx 180 ry 0 rz 180 deg; joints [-18.013, 9.38, 64.252, 49.087, 24.154, -46.475]
  Call Extruder(199.43818)
  MoveL 5025 to (229.18, 36.07, 78.65) mm, rotated rx 180 ry 0 rz 180 deg; joints [-18.01, 9.417, 64.21, 49.073, 24.157, -46.461]
  MoveL 5026 to (229.18, 36.07, 78.65) mm, rotated rx 180 ry 0 rz 180 deg; joints [-18.01, 9.417, 64.21, 49.073, 24.157, -46.461]
  Call Extruder(199.55280)
  MoveL 5027 to (229.38, 36.12, 78.65) mm, rotated rx -180 ry 0 rz 180 deg; joints [-18.008, 9.453, 64.167, 49.059, 24.159, -46.446]
  MoveL 5028 to (229.38, 36.12, 78.65) mm, rotated rx -180 ry 0 rz 180 deg; joints [-18.008, 9.453, 64.167, 49.059, 24.159, -46.446]
  Call Extruder(199.66788)
  MoveL 5029 to (229.59, 36.16, 78.65) mm, rotated rx 180 ry 0 rz 180 deg; joints [-18.006, 9.489, 64.125, 49.044, 24.161, -46.431]
  MoveL 5030 to (229.59, 36.16, 78.65) mm, rotated rx 180 ry 0 rz 180 deg; joints [-18.006, 9.489, 64.125, 49.044, 24.161, -46.431]
  Call Extruder(199.79011)
  MoveL 5031 to (229.8, 36.22, 78.65) mm, rotated rx 180 ry 0 rz 180 deg; joints [-18.004, 9.528, 64.08, 49.031, 24.164, -46.417]
  MoveL 5032 to (229.8, 36.22, 78.65) mm, rotated rx 180 ry 0 rz 180 deg; joints [-18.004, 9.528, 64.08, 49.031, 24.164, -46.417]
  Call Extruder(199.91978)
  MoveL 5033 to (230.02, 36.28, 78.65) mm, rotated rx -180 ry 0 rz -180 deg; joints [-18.004, 9.569, 64.032, 49.019, 24.168, -46.403]
  MoveL 5034 to (230.02, 36.28, 78.65) mm, rotated rx -180 ry 0 rz -180 deg; joints [-18.004, 9.569, 64.032, 49.019, 24.168, -46.403]
  Call Extruder(200.05001)
  MoveL 5035 to (230.25, 36.35, 78.65) mm, rotated rx 180 ry 0 rz 180 deg; joints [-18.003, 9.61, 63.984, 49.006, 24.172, -46.39]
  MoveL 5036 to (230.25, 36.35, 78.65) mm, rotated rx 180 ry 0 rz 180 deg; joints [-18.003, 9.61, 63.984, 49.006, 24.172, -46.39]
  Call Extruder(200.18080)
  MoveL 5037 to (230.47, 36.42, 78.65) mm, rotated rx -180 ry 0 rz 180 deg; joints [-18.003, 9.651, 63.936, 48.994, 24.176, -46.376]
  MoveL 5038 to (230.47, 36.42, 78.65) mm, rotated rx -180 ry 0 rz 180 deg; joints [-18.003, 9.651, 63.936, 48.994, 24.176, -46.376]
  Call Extruder(200.31217)
  MoveL 5039 to (230.69, 36.49, 78.65) mm, rotated rx 180 ry 0 rz 180 deg; joints [-18.002, 9.692, 63.888, 48.981, 24.181, -46.363]
  MoveL 5040 to (230.69, 36.49, 78.65) mm, rotated rx 180 ry 0 rz 180 deg; joints [-18.002, 9.692, 63.888, 48.981, 24.181, -46.363]
  Call Extruder(200.42119)
  MoveL 5041 to (230.88, 36.55, 78.65) mm, rotated rx -180 ry 0 rz -180 deg; joints [-18.002, 9.726, 63.848, 48.972, 24.184, -46.352]
  MoveL 5042 to (230.88, 36.55, 78.65) mm, rotated rx -180 ry 0 rz -180 deg; joints [-18.002, 9.726, 63.848, 48.972, 24.184, -46.352]
  Call Extruder(200.53270)
  MoveL 5043 to (231.06, 36.61, 78.65) mm, rotated rx 180 ry 0 rz 180 deg; joints [-18.002, 9.761, 63.808, 48.962, 24.188, -46.341]
  MoveL 5044 to (231.06, 36.61, 78.65) mm, rotated rx 180 ry 0 rz 180 deg; joints [-18.002, 9.761, 63.808, 48.962, 24.188, -46.341]
  Call Extruder(200.64671)
  MoveL 5045 to (231.26, 36.67, 78.65) mm, rotated rx 180 ry 0 rz 180 deg; joints [-18.002, 9.796, 63.766, 48.951, 24.192, -46.33]
  MoveL 5046 to (231.26, 36.67, 78.65) mm, rotated rx 180 ry 0 rz 180 deg; joints [-18.002, 9.796, 63.766, 48.951, 24.192, -46.33]
  Call Extruder(200.76118)
  MoveL 5047 to (231.45, 36.73, 78.65) mm, rotated rx 180 ry 0 rz 180 deg; joints [-18.002, 9.832, 63.725, 48.941, 24.196, -46.319]
  MoveL 5048 to (231.45, 36.73, 78.65) mm, rotated rx 180 ry 0 rz 180 deg; joints [-18.002, 9.832, 63.725, 48.941, 24.196, -46.319]
  Call Extruder(200.87611)
  MoveL 5049 to (231.64, 36.79, 78.65) mm, rotated rx 180 ry 0 rz 180 deg; joints [-18.002, 9.867, 63.684, 48.931, 24.2, -46.308]
  MoveL 5050 to (231.64, 36.79, 78.65) mm, rotated rx 180 ry 0 rz 180 deg; joints [-18.002, 9.867, 63.684, 48.931, 24.2, -46.308]
  Call Extruder(201.05806)
  MoveL 5051 to (231.93, 36.91, 78.65) mm, rotated rx -180 ry 0 rz -180 deg; joints [-18.005, 9.922, 63.619, 48.92, 24.208, -46.295]
  MoveL 5052 to (231.93, 36.91, 78.65) mm, rotated rx -180 ry 0 rz -180 deg; joints [-18.005, 9.922, 63.619, 48.92, 24.208, -46.295]
  Call Extruder(201.24078)
  MoveL 5053 to (232.22, 37.04, 78.65) mm, rotated rx 180 ry 0 rz 180 deg; joints [-18.008, 9.978, 63.553, 48.908, 24.217, -46.281]
  MoveL 5054 to (232.22, 37.04, 78.65) mm, rotated rx 180 ry 0 rz 180 deg; joints [-18.008, 9.978, 63.553, 48.908, 24.217, -46.281]
  Call Extruder(201.41120)
  MoveL 5055 to (232.49, 37.15, 78.65) mm, rotated rx -180 ry 0 rz 180 deg; joints [-18.011, 10.03, 63.493, 48.898, 24.225, -46.269]
  MoveL 5056 to (232.49, 37.15, 78.65) mm, rotated rx -180 ry 0 rz 180 deg; joints [-18.011, 10.03, 63.493, 48.898, 24.225, -46.269]
  Call Extruder(201.56919)
  MoveL 5057 to (232.74, 37.26, 78.65) mm, rotated rx 180 ry 0 rz 180 deg; joints [-18.013, 10.077, 63.437, 48.889, 24.232, -46.258]
  MoveL 5058 to (232.74, 37.26, 78.65) mm, rotated rx 180 ry 0 rz 180 deg; joints [-18.013, 10.077, 63.437, 48.889, 24.232, -46.258]
  Call Extruder(201.72780)
  MoveL 5059 to (232.99, 37.36, 78.65) mm, rotated rx 180 ry 0 rz -180 deg; joints [-18.016, 10.125, 63.38, 48.879, 24.24, -46.247]
  MoveL 5060 to (232.99, 37.36, 78.65) mm, rotated rx 180 ry 0 rz -180 deg; joints [-18.016, 10.125, 63.38, 48.879, 24.24, -46.247]
  Call Extruder(201.93396)
  MoveL 5061 to (233.29, 37.54, 78.65) mm, rotated rx -180 ry 0 rz 180 deg; joints [-18.024, 10.186, 63.309, 48.875, 24.253, -46.24]
  MoveL 5062 to (233.29, 37.54, 78.65) mm, rotated rx -180 ry 0 rz 180 deg; joints [-18.024, 10.186, 63.309, 48.875, 24.253, -46.24]
  Call Extruder(202.14091)
  MoveL 5063 to (233.6, 37.71, 78.65) mm, rotated rx 180 ry 0 rz 180 deg; joints [-18.033, 10.247, 63.237, 48.871, 24.266, -46.233]
  MoveL 5064 to (233.6, 37.71, 78.65) mm, rotated rx 180 ry 0 rz 180 deg; joints [-18.033, 10.247, 63.237, 48.871, 24.266, -46.233]
  Call Extruder(202.34863)
  MoveL 5065 to (233.9, 37.89, 78.65) mm, rotated rx -180 ry 0 rz -180 deg; joints [-18.041, 10.308, 63.165, 48.867, 24.279, -46.225]
  MoveL 5066 to (233.9, 37.89, 78.65) mm, rotated rx -180 ry 0 rz -180 deg; joints [-18.041, 10.308, 63.165, 48.867, 24.279, -46.225]
  Call Extruder(202.55713)
  MoveL 5067 to (234.21, 38.07, 78.65) mm, rotated rx 180 ry 0 rz -180 deg; joints [-18.049, 10.369, 63.093, 48.862, 24.293, -46.218]
  MoveL 5068 to (234.21, 38.07, 78.65) mm, rotated rx 180 ry 0 rz -180 deg; joints [-18.049, 10.369, 63.093, 48.862, 24.293, -46.218]
  Call Extruder(202.73668)
  MoveL 5069 to (234.45, 38.24, 78.65) mm, rotated rx 180 ry 0 rz 180 deg; joints [-18.06, 10.42, 63.033, 48.864, 24.306, -46.217]
  MoveL 5070 to (234.45, 38.24, 78.65) mm, rotated rx 180 ry 0 rz 180 deg; joints [-18.06, 10.42, 63.033, 48.864, 24.306, -46.217]
  Call Extruder(203.07009)
  MoveL 5071 to (234.9, 38.57, 78.65) mm, rotated rx 180 ry 0 rz 180 deg; joints [-18.079, 10.514, 62.921, 48.868, 24.332, -46.215]
  MoveL 5072 to (234.9, 38.57, 78.65) mm, rotated rx 180 ry 0 rz 180 deg; joints [-18.079, 10.514, 62.921, 48.868, 24.332, -46.215]
  Call Extruder(203.40469)
  MoveL 5073 to (235.35, 38.9, 78.65) mm, rotated rx 180 ry 0 rz 180 deg; joints [-18.099, 10.609, 62.809, 48.872, 24.357, -46.213]
  Call Extruder(204.23264)
  MoveL 5074 to (236.39, 39.81, 78.65) mm, rotated rx 180 ry 0 rz -180 deg; joints [-18.16, 10.836, 62.54, 48.905, 24.43, -46.23]
  Call Extruder(205.06059)
  MoveL 5075 to (237.3, 40.85, 78.65) mm, rotated rx 180 ry 0 rz 180 deg; joints [-18.24, 11.049, 62.286, 48.969, 24.514, -46.276]
  Call Extruder(205.22789)
  MoveL 5076 to (237.47, 41.07, 78.65) mm, rotated rx -180 ry 0 rz 180 deg; joints [-18.258, 11.09, 62.237, 48.987, 24.532, -46.289]
  MoveL 5077 to (237.47, 41.07, 78.65) mm, rotated rx -180 ry 0 rz 180 deg; joints [-18.258, 11.09, 62.237, 48.987, 24.532, -46.289]
  Call Extruder(205.56130)
  MoveL 5078 to (237.79, 41.52, 78.65) mm, rotated rx 180 ry 0 rz 180 deg; joints [-18.295, 11.171, 62.14, 49.022, 24.569, -46.316]
  MoveL 5079 to (237.79, 41.52, 78.65) mm, rotated rx 180 ry 0 rz 180 deg; joints [-18.295, 11.171, 62.14, 49.022, 24.569, -46.316]
  Call Extruder(205.89353)
  MoveL 5080 to (238.12, 41.97, 78.65) mm, rotated rx -180 ry 0 rz 180 deg; joints [-18.332, 11.253, 62.042, 49.057, 24.606, -46.342]
  MoveL 5081 to (238.12, 41.97, 78.65) mm, rotated rx -180 ry 0 rz 180 deg; joints [-18.332, 11.253, 62.042, 49.057, 24.606, -46.342]
  Call Extruder(206.01123)
  MoveL 5082 to (238.22, 42.15, 78.65) mm, rotated rx 180 ry 0 rz 180 deg; joints [-18.346, 11.28, 62.01, 49.072, 24.62, -46.355]
  MoveL 5083 to (238.22, 42.15, 78.65) mm, rotated rx 180 ry 0 rz 180 deg; joints [-18.346, 11.28, 62.01, 49.072, 24.62, -46.355]
  Call Extruder(206.21895)
  MoveL 5084 to (238.4, 42.45, 78.65) mm, rotated rx 180 ry 0 rz 180 deg; joints [-18.373, 11.327, 61.953, 49.1, 24.646, -46.378]
  MoveL 5085 to (238.4, 42.45, 78.65) mm, rotated rx 180 ry 0 rz 180 deg; joints [-18.373, 11.327, 61.953, 49.1, 24.646, -46.378]
  Call Extruder(206.42590)
  MoveL 5086 to (238.57, 42.75, 78.65) mm, rotated rx 180 ry 0 rz 180 deg; joints [-18.399, 11.374, 61.897, 49.128, 24.671, -46.4]
  MoveL 5087 to (238.57, 42.75, 78.65) mm, rotated rx 180 ry 0 rz 180 deg; joints [-18.399, 11.374, 61.897, 49.128, 24.671, -46.4]
  Call Extruder(206.63206)
  MoveL 5088 to (238.75, 43.06, 78.65) mm, rotated rx 180 ry 0 rz 180 deg; joints [-18.425, 11.421, 61.84, 49.156, 24.696, -46.422]
  MoveL 5089 to (238.75, 43.06, 78.65) mm, rotated rx 180 ry 0 rz 180 deg; joints [-18.425, 11.421, 61.84, 49.156, 24.696, -46.422]
  Call Extruder(206.81375)
  MoveL 5090 to (238.89, 43.34, 78.65) mm, rotated rx 180 ry 0 rz 180 deg; joints [-18.45, 11.462, 61.792, 49.183, 24.719, -46.445]
  MoveL 5091 to (238.89, 43.34, 78.65) mm, rotated rx 180 ry 0 rz 180 deg; joints [-18.45, 11.462, 61.792, 49.183, 24.719, -46.445]
  Call Extruder(206.97176)
  MoveL 5092 to (239, 43.58, 78.65) mm, rotated rx -180 ry 0 rz 180 deg; joints [-18.472, 11.494, 61.753, 49.21, 24.74, -46.467]
  MoveL 5093 to (239, 43.58, 78.65) mm, rotated rx -180 ry 0 rz 180 deg; joints [-18.472, 11.494, 61.753, 49.21, 24.74, -46.467]
  Call Extruder(207.12917)
  MoveL 5094 to (239.11, 43.83, 78.65) mm, rotated rx 180 ry 0 rz -180 deg; joints [-18.495, 11.527, 61.713, 49.237, 24.76, -46.489]
  MoveL 5095 to (239.11, 43.83, 78.65) mm, rotated rx 180 ry 0 rz -180 deg; joints [-18.495, 11.527, 61.713, 49.237, 24.76, -46.489]
  Call Extruder(207.31188)
  MoveL 5096 to (239.23, 44.13, 78.65) mm, rotated rx 180 ry 0 rz 180 deg; joints [-18.522, 11.564, 61.668, 49.268, 24.785, -46.515]
  MoveL 5097 to (239.23, 44.13, 78.65) mm, rotated rx 180 ry 0 rz 180 deg; joints [-18.522, 11.564, 61.668, 49.268, 24.785, -46.515]
  Call Extruder(207.49384)
  MoveL 5098 to (239.35, 44.42, 78.65) mm, rotated rx 180 ry 0 rz 180 deg; joints [-18.549, 11.602, 61.623, 49.3, 24.809, -46.541]
  MoveL 5099 to (239.35, 44.42, 78.65) mm, rotated rx 180 ry 0 rz 180 deg; joints [-18.549, 11.602, 61.623, 49.3, 24.809, -46.541]
  Call Extruder(207.64117)
  MoveL 5100 to (239.44, 44.66, 78.65) mm, rotated rx 180 ry 0 rz 180 deg; joints [-18.571, 11.631, 61.588, 49.327, 24.829, -46.564]
  MoveL 5101 to (239.44, 44.66, 78.65) mm, rotated rx 180 ry 0 rz 180 deg; joints [-18.571, 11.631, 61.588, 49.327, 24.829, -46.564]
  Call Extruder(207.75441)
  MoveL 5102 to (239.5, 44.85, 78.65) mm, rotated rx -180 ry 0 rz 180 deg; joints [-18.589, 11.653, 61.562, 49.349, 24.845, -46.582]
  MoveL 5103 to (239.5, 44.85, 78.65) mm, rotated rx -180 ry 0 rz 180 deg; joints [-18.589, 11.653, 61.562, 49.349, 24.845, -46.582]
  Call Extruder(207.86720)
  MoveL 5104 to (239.56, 45.03, 78.65) mm, rotated rx 180 ry 0 rz -180 deg; joints [-18.607, 11.674, 61.536, 49.371, 24.861, -46.601]
  MoveL 5105 to (239.56, 45.03, 78.65) mm, rotated rx 180 ry 0 rz -180 deg; joints [-18.607, 11.674, 61.536, 49.371, 24.861, -46.601]
  Call Extruder(207.97954)
  MoveL 5106 to (239.62, 45.22, 78.65) mm, rotated rx -180 ry 0 rz -180 deg; joints [-18.625, 11.696, 61.51, 49.393, 24.877, -46.62]
  MoveL 5107 to (239.62, 45.22, 78.65) mm, rotated rx -180 ry 0 rz -180 deg; joints [-18.625, 11.696, 61.51, 49.393, 24.877, -46.62]
  Call Extruder(208.09145)
  MoveL 5108 to (239.68, 45.41, 78.65) mm, rotated rx 180 ry 0 rz 180 deg; joints [-18.642, 11.717, 61.485, 49.415, 24.893, -46.638]
  MoveL 5109 to (239.68, 45.41, 78.65) mm, rotated rx 180 ry 0 rz 180 deg; joints [-18.642, 11.717, 61.485, 49.415, 24.893, -46.638]
  Call Extruder(208.21285)
  MoveL 5110 to (239.75, 45.62, 78.65) mm, rotated rx -180 ry 0 rz 180 deg; joints [-18.662, 11.74, 61.457, 49.439, 24.91, -46.658]
  MoveL 5111 to (239.75, 45.62, 78.65) mm, rotated rx -180 ry 0 rz 180 deg; joints [-18.662, 11.74, 61.457, 49.439, 24.91, -46.658]
  Call Extruder(208.34364)
  MoveL 5112 to (239.82, 45.84, 78.65) mm, rotated rx 180 ry 0 rz 180 deg; joints [-18.683, 11.765, 61.427, 49.465, 24.929, -46.681]
  MoveL 5113 to (239.82, 45.84, 78.65) mm, rotated rx 180 ry 0 rz 180 deg; joints [-18.683, 11.765, 61.427, 49.465, 24.929, -46.681]
  Call Extruder(208.47386)
  MoveL 5114 to (239.88, 46.06, 78.65) mm, rotated rx -180 ry 0 rz 180 deg; joints [-18.705, 11.789, 61.397, 49.492, 24.948, -46.703]
  MoveL 5115 to (239.88, 46.06, 78.65) mm, rotated rx -180 ry 0 rz 180 deg; joints [-18.705, 11.789, 61.397, 49.492, 24.948, -46.703]
  Call Extruder(208.60352)
  MoveL 5116 to (239.95, 46.29, 78.65) mm, rotated rx -180 ry 0 rz 180 deg; joints [-18.726, 11.814, 61.367, 49.518, 24.966, -46.725]
  MoveL 5117 to (239.95, 46.29, 78.65) mm, rotated rx -180 ry 0 rz 180 deg; joints [-18.726, 11.814, 61.367, 49.518, 24.966, -46.725]
  Call Extruder(208.73262)
  MoveL 5118 to (240.02, 46.51, 78.65) mm, rotated rx 180 ry 0 rz 180 deg; joints [-18.747, 11.839, 61.338, 49.544, 24.985, -46.747]
  MoveL 5119 to (240.02, 46.51, 78.65) mm, rotated rx 180 ry 0 rz 180 deg; joints [-18.747, 11.839, 61.338, 49.544, 24.985, -46.747]
  Call Extruder(208.84768)
  MoveL 5120 to (240.06, 46.72, 78.65) mm, rotated rx -180 ry 0 rz 180 deg; joints [-18.767, 11.858, 61.314, 49.57, 25.002, -46.77]
  MoveL 5121 to (240.06, 46.72, 78.65) mm, rotated rx -180 ry 0 rz 180 deg; joints [-18.767, 11.858, 61.314, 49.57, 25.002, -46.77]
  Call Extruder(208.96228)
  MoveL 5122 to (240.11, 46.92, 78.65) mm, rotated rx 180 ry 0 rz -180 deg; joints [-18.787, 11.878, 61.29, 49.596, 25.02, -46.792]
  MoveL 5123 to (240.11, 46.92, 78.65) mm, rotated rx 180 ry 0 rz -180 deg; joints [-18.787, 11.878, 61.29, 49.596, 25.02, -46.792]
  Call Extruder(209.07643)
  MoveL 5124 to (240.15, 47.12, 78.65) mm, rotated rx -180 ry 0 rz 180 deg; joints [-18.807, 11.898, 61.267, 49.622, 25.037, -46.814]
  MoveL 5125 to (240.15, 47.12, 78.65) mm, rotated rx -180 ry 0 rz 180 deg; joints [-18.807, 11.898, 61.267, 49.622, 25.037, -46.814]
  Call Extruder(209.19012)
  MoveL 5126 to (240.2, 47.33, 78.65) mm, rotated rx 180 ry 0 rz 180 deg; joints [-18.827, 11.917, 61.243, 49.647, 25.054, -46.836]
  MoveL 5127 to (240.2, 47.33, 78.65) mm, rotated rx 180 ry 0 rz 180 deg; joints [-18.827, 11.917, 61.243, 49.647, 25.054, -46.836]
  Call Extruder(209.31554)
  MoveL 5128 to (240.24, 47.55, 78.65) mm, rotated rx 180 ry 0 rz 180 deg; joints [-18.85, 11.939, 61.217, 49.676, 25.073, -46.86]
  MoveL 5129 to (240.24, 47.55, 78.65) mm, rotated rx 180 ry 0 rz 180 deg; joints [-18.85, 11.939, 61.217, 49.676, 25.073, -46.86]
  Call Extruder(209.45251)
  MoveL 5130 to (240.29, 47.8, 78.65) mm, rotated rx 180 ry 0 rz -180 deg; joints [-18.874, 11.962, 61.189, 49.708, 25.094, -46.887]
  MoveL 5131 to (240.29, 47.8, 78.65) mm, rotated rx 180 ry 0 rz -180 deg; joints [-18.874, 11.962, 61.189, 49.708, 25.094, -46.887]
  Call Extruder(209.58888)
  MoveL 5132 to (240.34, 48.05, 78.65) mm, rotated rx -180 ry 0 rz 180 deg; joints [-18.899, 11.985, 61.161, 49.739, 25.116, -46.914]
  MoveL 5133 to (240.34, 48.05, 78.65) mm, rotated rx -180 ry 0 rz 180 deg; joints [-18.899, 11.985, 61.161, 49.739, 25.116, -46.914]
  Call Extruder(209.72464)
  MoveL 5134 to (240.39, 48.3, 78.65) mm, rotated rx -180 ry 0 rz 180 deg; joints [-18.923, 12.009, 61.132, 49.771, 25.137, -46.941]
  MoveL 5135 to (240.39, 48.3, 78.65) mm, rotated rx -180 ry 0 rz 180 deg; joints [-18.923, 12.009, 61.132, 49.771, 25.137, -46.941]
  Call Extruder(209.85978)
  MoveL 5136 to (240.44, 48.55, 78.65) mm, rotated rx -180 ry 0 rz 180 deg; joints [-18.948, 12.032, 61.104, 49.802, 25.158, -46.968]
  MoveL 5137 to (240.44, 48.55, 78.65) mm, rotated rx -180 ry 0 rz 180 deg; joints [-18.948, 12.032, 61.104, 49.802, 25.158, -46.968]
  Call Extruder(209.99432)
  MoveL 5138 to (240.49, 48.8, 78.65) mm, rotated rx 180 ry 0 rz 180 deg; joints [-18.973, 12.055, 61.076, 49.834, 25.179, -46.995]
  MoveL 5139 to (240.49, 48.8, 78.65) mm, rotated rx 180 ry 0 rz 180 deg; joints [-18.973, 12.055, 61.076, 49.834, 25.179, -46.995]
  Call Extruder(210.12825)
  MoveL 5140 to (240.54, 49.05, 78.65) mm, rotated rx -180 ry 0 rz -180 deg; joints [-18.997, 12.078, 61.048, 49.865, 25.2, -47.022]
  MoveL 5141 to (240.54, 49.05, 78.65) mm, rotated rx -180 ry 0 rz -180 deg; joints [-18.997, 12.078, 61.048, 49.865, 25.2, -47.022]
  Call Extruder(210.27611)
  MoveL 5142 to (240.59, 49.33, 78.65) mm, rotated rx -180 ry 0 rz 180 deg; joints [-19.025, 12.103, 61.018, 49.9, 25.223, -47.052]
  MoveL 5143 to (240.59, 49.33, 78.65) mm, rotated rx -180 ry 0 rz 180 deg; joints [-19.025, 12.103, 61.018, 49.9, 25.223, -47.052]
  Call Extruder(210.43786)
  MoveL 5144 to (240.64, 49.63, 78.65) mm, rotated rx 180 ry 0 rz 180 deg; joints [-19.055, 12.13, 60.985, 49.94, 25.249, -47.086]
  MoveL 5145 to (240.64, 49.63, 78.65) mm, rotated rx 180 ry 0 rz 180 deg; joints [-19.055, 12.13, 60.985, 49.94, 25.249, -47.086]
  Call Extruder(210.59887)
  MoveL 5146 to (240.69, 49.94, 78.65) mm, rotated rx -180 ry 0 rz 180 deg; joints [-19.086, 12.157, 60.953, 49.98, 25.275, -47.12]
  MoveL 5147 to (240.69, 49.94, 78.65) mm, rotated rx -180 ry 0 rz 180 deg; joints [-19.086, 12.157, 60.953, 49.98, 25.275, -47.12]
  Call Extruder(210.75916)
  MoveL 5148 to (240.74, 50.24, 78.65) mm, rotated rx 180 ry 0 rz 180 deg; joints [-19.116, 12.183, 60.921, 50.019, 25.301, -47.154]
  MoveL 5149 to (240.74, 50.24, 78.65) mm, rotated rx 180 ry 0 rz 180 deg; joints [-19.116, 12.183, 60.921, 50.019, 25.301, -47.154]
  Call Extruder(210.91872)
  MoveL 5150 to (240.78, 50.55, 78.65) mm, rotated rx -180 ry 0 rz -180 deg; joints [-19.146, 12.21, 60.888, 50.058, 25.327, -47.187]
  MoveL 5151 to (240.78, 50.55, 78.65) mm, rotated rx -180 ry 0 rz -180 deg; joints [-19.146, 12.21, 60.888, 50.058, 25.327, -47.187]
  Call Extruder(211.07756)
  MoveL 5152 to (240.83, 50.86, 78.65) mm, rotated rx -180 ry 0 rz -180 deg; joints [-19.177, 12.237, 60.856, 50.097, 25.353, -47.221]
  MoveL 5153 to (240.83, 50.86, 78.65) mm, rotated rx -180 ry 0 rz -180 deg; joints [-19.177, 12.237, 60.856, 50.097, 25.353, -47.221]
  Call Extruder(211.25623)
  MoveL 5154 to (240.88, 51.2, 78.65) mm, rotated rx 180 ry 0 rz 180 deg; joints [-19.212, 12.266, 60.821, 50.142, 25.383, -47.259]
  MoveL 5155 to (240.88, 51.2, 78.65) mm, rotated rx 180 ry 0 rz 180 deg; joints [-19.212, 12.266, 60.821, 50.142, 25.383, -47.259]
  Call Extruder(211.45467)
  MoveL 5156 to (240.92, 51.59, 78.65) mm, rotated rx -180 ry 0 rz 180 deg; joints [-19.251, 12.297, 60.783, 50.193, 25.416, -47.303]
  MoveL 5157 to (240.92, 51.59, 78.65) mm, rotated rx -180 ry 0 rz 180 deg; joints [-19.251, 12.297, 60.783, 50.193, 25.416, -47.303]
  Call Extruder(211.65225)
  MoveL 5158 to (240.97, 51.98, 78.65) mm, rotated rx 180 ry 0 rz -180 deg; joints [-19.29, 12.328, 60.744, 50.244, 25.449, -47.347]
  MoveL 5159 to (240.97, 51.98, 78.65) mm, rotated rx 180 ry 0 rz -180 deg; joints [-19.29, 12.328, 60.744, 50.244, 25.449, -47.347]
  Call Extruder(211.84895)
  MoveL 5160 to (241.02, 52.36, 78.65) mm, rotated rx -180 ry 0 rz 180 deg; joints [-19.329, 12.36, 60.706, 50.294, 25.482, -47.39]
  MoveL 5161 to (241.02, 52.36, 78.65) mm, rotated rx -180 ry 0 rz 180 deg; joints [-19.329, 12.36, 60.706, 50.294, 25.482, -47.39]
  Call Extruder(212.04479)
  MoveL 5162 to (241.06, 52.75, 78.65) mm, rotated rx 180 ry 0 rz 180 deg; joints [-19.368, 12.391, 60.668, 50.345, 25.515, -47.433]
  MoveL 5163 to (241.06, 52.75, 78.65) mm, rotated rx 180 ry 0 rz 180 deg; joints [-19.368, 12.391, 60.668, 50.345, 25.515, -47.433]
  Call Extruder(212.34023)
  MoveL 5164 to (241.11, 53.34, 78.65) mm, rotated rx -180 ry 0 rz 180 deg; joints [-19.428, 12.435, 60.614, 50.424, 25.566, -47.501]
  MoveL 5165 to (241.11, 53.34, 78.65) mm, rotated rx -180 ry 0 rz 180 deg; joints [-19.428, 12.435, 60.614, 50.424, 25.566, -47.501]
  Call Extruder(212.63433)
  MoveL 5166 to (241.15, 53.93, 78.65) mm, rotated rx -180 ry 0 rz 180 deg; joints [-19.488, 12.479, 60.561, 50.502, 25.616, -47.569]
  MoveL 5167 to (241.15, 53.93, 78.65) mm, rotated rx -180 ry 0 rz 180 deg; joints [-19.488, 12.479, 60.561, 50.502, 25.616, -47.569]
  Call Extruder(212.92711)
  MoveL 5168 to (241.2, 54.52, 78.65) mm, rotated rx 180 ry 0 rz 180 deg; joints [-19.548, 12.524, 60.507, 50.58, 25.667, -47.636]
  MoveL 5169 to (241.2, 54.52, 78.65) mm, rotated rx 180 ry 0 rz 180 deg; joints [-19.548, 12.524, 60.507, 50.58, 25.667, -47.636]
  Call Extruder(213.50056)
  MoveL 5170 to (241.25, 55.68, 78.65) mm, rotated rx -180 ry 0 rz 180 deg; joints [-19.668, 12.604, 60.409, 50.738, 25.766, -47.772]
  MoveL 5171 to (241.25, 55.68, 78.65) mm, rotated rx -180 ry 0 rz 180 deg; joints [-19.668, 12.604, 60.409, 50.738, 25.766, -47.772]
  Call Extruder(214.21439)
  MoveL 5172 to (241.29, 57.14, 78.65) mm, rotated rx -180 ry 0 rz 180 deg; joints [-19.819, 12.701, 60.291, 50.935, 25.892, -47.943]
  Call Extruder(256.27928)
  MoveL 5173 to (241.29, 142.86, 78.65) mm, rotated rx 180 ry 0 rz 180 deg; joints [-28.232, 19.602, 51.431, 58.81, 33.571, -53.999]
  Call Extruder(256.70771)
  MoveL 5174 to (241.27, 143.73, 78.65) mm, rotated rx -180 ry 0 rz 180 deg; joints [-28.313, 19.687, 51.316, 58.858, 33.652, -54.025]
  MoveL 5175 to (241.27, 143.73, 78.65) mm, rotated rx -180 ry 0 rz 180 deg; joints [-28.313, 19.687, 51.316, 58.858, 33.652, -54.025]
  Call Extruder(257.28116)
  MoveL 5176 to (241.22, 144.9, 78.65) mm, rotated rx 180 ry 0 rz -180 deg; joints [-28.421, 19.796, 51.168, 58.924, 33.759, -54.061]
  MoveL 5177 to (241.22, 144.9, 78.65) mm, rotated rx 180 ry 0 rz -180 deg; joints [-28.421, 19.796, 51.168, 58.924, 33.759, -54.061]
  Call Extruder(257.71549)
  MoveL 5178 to (241.18, 145.77, 78.65) mm, rotated rx 180 ry 0 rz 180 deg; joints [-28.503, 19.877, 51.059, 58.974, 33.84, -54.089]
  MoveL 5179 to (241.18, 145.77, 78.65) mm, rotated rx 180 ry 0 rz 180 deg; joints [-28.503, 19.877, 51.059, 58.974, 33.84, -54.089]
  Call Extruder(258.00960)
  MoveL 5180 to (241.13, 146.36, 78.65) mm, rotated rx 180 ry 0 rz 180 deg; joints [-28.559, 19.929, 50.989, 59.01, 33.895, -54.11]
  MoveL 5181 to (241.13, 146.36, 78.65) mm, rotated rx 180 ry 0 rz 180 deg; joints [-28.559, 19.929, 50.989, 59.01, 33.895, -54.11]
  Call Extruder(258.30504)
  MoveL 5182 to (241.09, 146.95, 78.65) mm, rotated rx -180 ry 0 rz 180 deg; joints [-28.615, 19.981, 50.919, 59.045, 33.95, -54.131]
  MoveL 5183 to (241.09, 146.95, 78.65) mm, rotated rx -180 ry 0 rz 180 deg; joints [-28.615, 19.981, 50.919, 59.045, 33.95, -54.131]
  Call Extruder(258.55130)
  MoveL 5184 to (241.04, 147.44, 78.65) mm, rotated rx 180 ry 0 rz 180 deg; joints [-28.662, 20.022, 50.862, 59.075, 33.995, -54.149]
  MoveL 5185 to (241.04, 147.44, 78.65) mm, rotated rx 180 ry 0 rz 180 deg; joints [-28.662, 20.022, 50.862, 59.075, 33.995, -54.149]
  Call Extruder(258.74800)
  MoveL 5186 to (240.99, 147.83, 78.65) mm, rotated rx -180 ry 0 rz 180 deg; joints [-28.7, 20.054, 50.82, 59.1, 34.032, -54.165]
  MoveL 5187 to (240.99, 147.83, 78.65) mm, rotated rx -180 ry 0 rz 180 deg; joints [-28.7, 20.054, 50.82, 59.1, 34.032, -54.165]
  Call Extruder(258.94558)
  MoveL 5188 to (240.95, 148.22, 78.65) mm, rotated rx 180 ry 0 rz 180 deg; joints [-28.737, 20.085, 50.777, 59.125, 34.068, -54.18]
  MoveL 5189 to (240.95, 148.22, 78.65) mm, rotated rx 180 ry 0 rz 180 deg; joints [-28.737, 20.085, 50.777, 59.125, 34.068, -54.18]
  Call Extruder(259.14402)
  MoveL 5190 to (240.9, 148.6, 78.65) mm, rotated rx -180 ry 0 rz 180 deg; joints [-28.774, 20.117, 50.734, 59.15, 34.104, -54.195]
  MoveL 5191 to (240.9, 148.6, 78.65) mm, rotated rx -180 ry 0 rz 180 deg; joints [-28.774, 20.117, 50.734, 59.15, 34.104, -54.195]
  Call Extruder(259.34333)
  MoveL 5192 to (240.86, 148.99, 78.65) mm, rotated rx -180 ry 0 rz -180 deg; joints [-28.812, 20.148, 50.692, 59.175, 34.14, -54.21]
  MoveL 5193 to (240.86, 148.99, 78.65) mm, rotated rx -180 ry 0 rz -180 deg; joints [-28.812, 20.148, 50.692, 59.175, 34.14, -54.21]
  Call Extruder(259.50216)
  MoveL 5194 to (240.81, 149.3, 78.65) mm, rotated rx -180 ry 0 rz -180 deg; joints [-28.842, 20.171, 50.661, 59.196, 34.168, -54.224]
  MoveL 5195 to (240.81, 149.3, 78.65) mm, rotated rx -180 ry 0 rz -180 deg; joints [-28.842, 20.171, 50.661, 59.196, 34.168, -54.224]
  Call Extruder(259.66172)
  MoveL 5196 to (240.76, 149.6, 78.65) mm, rotated rx 180 ry 0 rz -180 deg; joints [-28.872, 20.194, 50.63, 59.217, 34.197, -54.237]
  MoveL 5197 to (240.76, 149.6, 78.65) mm, rotated rx 180 ry 0 rz -180 deg; joints [-28.872, 20.194, 50.63, 59.217, 34.197, -54.237]
  Call Extruder(259.82201)
  MoveL 5198 to (240.71, 149.91, 78.65) mm, rotated rx 180 ry 0 rz -180 deg; joints [-28.902, 20.217, 50.599, 59.238, 34.226, -54.251]
  MoveL 5199 to (240.71, 149.91, 78.65) mm, rotated rx 180 ry 0 rz -180 deg; joints [-28.902, 20.217, 50.599, 59.238, 34.226, -54.251]
  Call Extruder(259.98302)
  MoveL 5200 to (240.66, 150.21, 78.65) mm, rotated rx 180 ry 0 rz -180 deg; joints [-28.932, 20.24, 50.568, 59.259, 34.254, -54.264]
  MoveL 5201 to (240.66, 150.21, 78.65) mm, rotated rx 180 ry 0 rz -180 deg; joints [-28.932, 20.24, 50.568, 59.259, 34.254, -54.264]
  Call Extruder(260.14477)
  MoveL 5202 to (240.61, 150.52, 78.65) mm, rotated rx 180 ry 0 rz 180 deg; joints [-28.962, 20.263, 50.537, 59.28, 34.283, -54.277]
  MoveL 5203 to (240.61, 150.52, 78.65) mm, rotated rx 180 ry 0 rz 180 deg; joints [-28.962, 20.263, 50.537, 59.28, 34.283, -54.277]
  Call Extruder(260.30724)
  MoveL 5204 to (240.57, 150.83, 78.65) mm, rotated rx 180 ry 0 rz 180 deg; joints [-28.993, 20.285, 50.506, 59.301, 34.311, -54.291]
  MoveL 5205 to (240.57, 150.83, 78.65) mm, rotated rx 180 ry 0 rz 180 deg; joints [-28.993, 20.285, 50.506, 59.301, 34.311, -54.291]
  Call Extruder(260.44117)
  MoveL 5206 to (240.52, 151.08, 78.65) mm, rotated rx 180 ry 0 rz 180 deg; joints [-29.017, 20.302, 50.483, 59.319, 34.335, -54.303]
  MoveL 5207 to (240.52, 151.08, 78.65) mm, rotated rx 180 ry 0 rz 180 deg; joints [-29.017, 20.302, 50.483, 59.319, 34.335, -54.303]
  Call Extruder(260.57570)
  MoveL 5208 to (240.47, 151.32, 78.65) mm, rotated rx 180 ry 0 rz 180 deg; joints [-29.043, 20.319, 50.46, 59.337, 34.358, -54.315]
  MoveL 5209 to (240.47, 151.32, 78.65) mm, rotated rx 180 ry 0 rz 180 deg; joints [-29.043, 20.319, 50.46, 59.337, 34.358, -54.315]
  Call Extruder(260.71085)
  MoveL 5210 to (240.42, 151.57, 78.65) mm, rotated rx 180 ry 0 rz 180 deg; joints [-29.067, 20.336, 50.437, 59.356, 34.382, -54.327]
  MoveL 5211 to (240.42, 151.57, 78.65) mm, rotated rx 180 ry 0 rz 180 deg; joints [-29.067, 20.336, 50.437, 59.356, 34.382, -54.327]
  Call Extruder(260.84661)
  MoveL 5212 to (240.37, 151.82, 78.65) mm, rotated rx 180 ry 0 rz 180 deg; joints [-29.092, 20.353, 50.414, 59.374, 34.405, -54.339]
  MoveL 5213 to (240.37, 151.82, 78.65) mm, rotated rx 180 ry 0 rz 180 deg; joints [-29.092, 20.353, 50.414, 59.374, 34.405, -54.339]
  Call Extruder(260.98297)
  MoveL 5214 to (240.32, 152.07, 78.65) mm, rotated rx 180 ry 0 rz 180 deg; joints [-29.117, 20.37, 50.391, 59.392, 34.428, -54.351]
  MoveL 5215 to (240.32, 152.07, 78.65) mm, rotated rx 180 ry 0 rz 180 deg; joints [-29.117, 20.37, 50.391, 59.392, 34.428, -54.351]
  Call Extruder(261.11995)
  MoveL 5216 to (240.27, 152.32, 78.65) mm, rotated rx 180 ry 0 rz 180 deg; joints [-29.142, 20.387, 50.368, 59.41, 34.452, -54.363]
  MoveL 5217 to (240.27, 152.32, 78.65) mm, rotated rx 180 ry 0 rz 180 deg; joints [-29.142, 20.387, 50.368, 59.41, 34.452, -54.363]
  Call Extruder(261.25754)
  MoveL 5218 to (240.22, 152.57, 78.65) mm, rotated rx -180 ry 0 rz -180 deg; joints [-29.167, 20.404, 50.345, 59.428, 34.475, -54.375]
  MoveL 5219 to (240.22, 152.57, 78.65) mm, rotated rx -180 ry 0 rz -180 deg; joints [-29.167, 20.404, 50.345, 59.428, 34.475, -54.375]
  Call Extruder(261.37124)
  MoveL 5220 to (240.17, 152.77, 78.65) mm, rotated rx 180 ry 0 rz 180 deg; joints [-29.188, 20.417, 50.327, 59.443, 34.494, -54.385]
  MoveL 5221 to (240.17, 152.77, 78.65) mm, rotated rx 180 ry 0 rz 180 deg; joints [-29.188, 20.417, 50.327, 59.443, 34.494, -54.385]
  Call Extruder(261.48539)
  MoveL 5222 to (240.13, 152.98, 78.65) mm, rotated rx 180 ry 0 rz -180 deg; joints [-29.209, 20.43, 50.309, 59.458, 34.514, -54.395]
  MoveL 5223 to (240.13, 152.98, 78.65) mm, rotated rx 180 ry 0 rz -180 deg; joints [-29.209, 20.43, 50.309, 59.458, 34.514, -54.395]
  Call Extruder(261.59999)
  MoveL 5224 to (240.08, 153.18, 78.65) mm, rotated rx 180 ry 0 rz -180 deg; joints [-29.229, 20.443, 50.291, 59.474, 34.533, -54.405]
  MoveL 5225 to (240.08, 153.18, 78.65) mm, rotated rx 180 ry 0 rz -180 deg; joints [-29.229, 20.443, 50.291, 59.474, 34.533, -54.405]
  Call Extruder(261.71505)
  MoveL 5226 to (240.04, 153.39, 78.65) mm, rotated rx -180 ry 0 rz 180 deg; joints [-29.25, 20.457, 50.273, 59.489, 34.552, -54.416]
  MoveL 5227 to (240.04, 153.39, 78.65) mm, rotated rx -180 ry 0 rz 180 deg; joints [-29.25, 20.457, 50.273, 59.489, 34.552, -54.416]
  Call Extruder(261.83727)
  MoveL 5228 to (239.98, 153.6, 78.65) mm, rotated rx 180 ry 0 rz 180 deg; joints [-29.272, 20.469, 50.256, 59.506, 34.572, -54.428]
  MoveL 5229 to (239.98, 153.6, 78.65) mm, rotated rx 180 ry 0 rz 180 deg; joints [-29.272, 20.469, 50.256, 59.506, 34.572, -54.428]
  Call Extruder(261.96693)
  MoveL 5230 to (239.92, 153.82, 78.65) mm, rotated rx 180 ry 0 rz 180 deg; joints [-29.296, 20.48, 50.241, 59.525, 34.593, -54.441]
  MoveL 5231 to (239.92, 153.82, 78.65) mm, rotated rx 180 ry 0 rz 180 deg; joints [-29.296, 20.48, 50.241, 59.525, 34.593, -54.441]
  Call Extruder(262.09716)
  MoveL 5232 to (239.85, 154.05, 78.65) mm, rotated rx -180 ry 0 rz 180 deg; joints [-29.319, 20.491, 50.227, 59.544, 34.615, -54.455]
  MoveL 5233 to (239.85, 154.05, 78.65) mm, rotated rx -180 ry 0 rz 180 deg; joints [-29.319, 20.491, 50.227, 59.544, 34.615, -54.455]
  Call Extruder(262.22795)
  MoveL 5234 to (239.78, 154.27, 78.65) mm, rotated rx 180 ry 0 rz 180 deg; joints [-29.343, 20.502, 50.211, 59.563, 34.636, -54.469]
  MoveL 5235 to (239.78, 154.27, 78.65) mm, rotated rx 180 ry 0 rz 180 deg; joints [-29.343, 20.502, 50.211, 59.563, 34.636, -54.469]
  Call Extruder(262.35930)
  MoveL 5236 to (239.71, 154.49, 78.65) mm, rotated rx 180 ry 0 rz -180 deg; joints [-29.366, 20.513, 50.196, 59.582, 34.657, -54.483]
  MoveL 5237 to (239.71, 154.49, 78.65) mm, rotated rx 180 ry 0 rz -180 deg; joints [-29.366, 20.513, 50.196, 59.582, 34.657, -54.483]
  Call Extruder(262.47120)
  MoveL 5238 to (239.65, 154.68, 78.65) mm, rotated rx 180 ry 0 rz 180 deg; joints [-29.386, 20.521, 50.185, 59.599, 34.675, -54.495]
  MoveL 5239 to (239.65, 154.68, 78.65) mm, rotated rx 180 ry 0 rz 180 deg; joints [-29.386, 20.521, 50.185, 59.599, 34.675, -54.495]
  Call Extruder(262.58355)
  MoveL 5240 to (239.59, 154.87, 78.65) mm, rotated rx 180 ry 0 rz 180 deg; joints [-29.406, 20.53, 50.173, 59.615, 34.693, -54.507]
  MoveL 5241 to (239.59, 154.87, 78.65) mm, rotated rx 180 ry 0 rz 180 deg; joints [-29.406, 20.53, 50.173, 59.615, 34.693, -54.507]
  Call Extruder(262.69634)
  MoveL 5242 to (239.53, 155.06, 78.65) mm, rotated rx 180 ry 0 rz -180 deg; joints [-29.426, 20.538, 50.162, 59.632, 34.711, -54.519]
  MoveL 5243 to (239.53, 155.06, 78.65) mm, rotated rx 180 ry 0 rz -180 deg; joints [-29.426, 20.538, 50.162, 59.632, 34.711, -54.519]
  Call Extruder(262.80957)
  MoveL 5244 to (239.47, 155.25, 78.65) mm, rotated rx -180 ry 0 rz -180 deg; joints [-29.446, 20.547, 50.15, 59.649, 34.728, -54.531]
  MoveL 5245 to (239.47, 155.25, 78.65) mm, rotated rx -180 ry 0 rz -180 deg; joints [-29.446, 20.547, 50.15, 59.649, 34.728, -54.531]
  Call Extruder(262.92325)
  MoveL 5246 to (239.41, 155.44, 78.65) mm, rotated rx -180 ry 0 rz -180 deg; joints [-29.466, 20.556, 50.138, 59.665, 34.746, -54.543]
  MoveL 5247 to (239.41, 155.44, 78.65) mm, rotated rx -180 ry 0 rz -180 deg; joints [-29.466, 20.556, 50.138, 59.665, 34.746, -54.543]
  Call Extruder(263.10521)
  MoveL 5248 to (239.29, 155.73, 78.65) mm, rotated rx 180 ry 0 rz -180 deg; joints [-29.499, 20.564, 50.127, 59.694, 34.774, -54.565]
  MoveL 5249 to (239.29, 155.73, 78.65) mm, rotated rx 180 ry 0 rz -180 deg; joints [-29.499, 20.564, 50.127, 59.694, 34.774, -54.565]
  Call Extruder(263.28793)
  MoveL 5250 to (239.16, 156.02, 78.65) mm, rotated rx -180 ry 0 rz 180 deg; joints [-29.531, 20.572, 50.115, 59.723, 34.802, -54.588]
  MoveL 5251 to (239.16, 156.02, 78.65) mm, rotated rx -180 ry 0 rz 180 deg; joints [-29.531, 20.572, 50.115, 59.723, 34.802, -54.588]
  Call Extruder(263.45835)
  MoveL 5252 to (239.05, 156.29, 78.65) mm, rotated rx 180 ry 0 rz 180 deg; joints [-29.561, 20.58, 50.105, 59.75, 34.828, -54.609]
  MoveL 5253 to (239.05, 156.29, 78.65) mm, rotated rx 180 ry 0 rz 180 deg; joints [-29.561, 20.58, 50.105, 59.75, 34.828, -54.609]
  Call Extruder(263.61637)
  MoveL 5254 to (238.94, 156.54, 78.65) mm, rotated rx 180 ry 0 rz 180 deg; joints [-29.589, 20.586, 50.096, 59.776, 34.852, -54.628]
  MoveL 5255 to (238.94, 156.54, 78.65) mm, rotated rx 180 ry 0 rz 180 deg; joints [-29.589, 20.586, 50.096, 59.776, 34.852, -54.628]
  Call Extruder(263.77499)
  MoveL 5256 to (238.84, 156.79, 78.65) mm, rotated rx -180 ry 0 rz -180 deg; joints [-29.617, 20.593, 50.087, 59.801, 34.876, -54.648]
  MoveL 5257 to (238.84, 156.79, 78.65) mm, rotated rx -180 ry 0 rz -180 deg; joints [-29.617, 20.593, 50.087, 59.801, 34.876, -54.648]
  Call Extruder(264.00155)
  MoveL 5258 to (238.65, 157.13, 78.65) mm, rotated rx 180 ry 0 rz 180 deg; joints [-29.656, 20.593, 50.086, 59.841, 34.908, -54.68]
  MoveL 5259 to (238.65, 157.13, 78.65) mm, rotated rx 180 ry 0 rz 180 deg; joints [-29.656, 20.593, 50.086, 59.841, 34.908, -54.68]
  Call Extruder(264.22896)
  MoveL 5260 to (238.46, 157.46, 78.65) mm, rotated rx -180 ry 0 rz 180 deg; joints [-29.696, 20.594, 50.085, 59.88, 34.941, -54.713]
  MoveL 5261 to (238.46, 157.46, 78.65) mm, rotated rx -180 ry 0 rz 180 deg; joints [-29.696, 20.594, 50.085, 59.88, 34.941, -54.713]
  Call Extruder(264.41617)
  MoveL 5262 to (238.3, 157.73, 78.65) mm, rotated rx 180 ry 0 rz 180 deg; joints [-29.729, 20.593, 50.087, 59.914, 34.967, -54.741]
  MoveL 5263 to (238.3, 157.73, 78.65) mm, rotated rx 180 ry 0 rz 180 deg; joints [-29.729, 20.593, 50.087, 59.914, 34.967, -54.741]
  Call Extruder(264.60408)
  MoveL 5264 to (238.13, 158.01, 78.65) mm, rotated rx -180 ry 0 rz -180 deg; joints [-29.761, 20.591, 50.089, 59.947, 34.994, -54.768]
  MoveL 5265 to (238.13, 158.01, 78.65) mm, rotated rx -180 ry 0 rz -180 deg; joints [-29.761, 20.591, 50.089, 59.947, 34.994, -54.768]
  Call Extruder(264.78361)
  MoveL 5266 to (237.96, 158.25, 78.65) mm, rotated rx 180 ry 0 rz 180 deg; joints [-29.792, 20.585, 50.098, 59.982, 35.018, -54.797]
  MoveL 5267 to (237.96, 158.25, 78.65) mm, rotated rx 180 ry 0 rz 180 deg; joints [-29.792, 20.585, 50.098, 59.982, 35.018, -54.797]
  Call Extruder(265.11703)
  MoveL 5268 to (237.63, 158.7, 78.65) mm, rotated rx 180 ry 0 rz 180 deg; joints [-29.849, 20.571, 50.116, 60.045, 35.062, -54.852]
  MoveL 5269 to (237.63, 158.7, 78.65) mm, rotated rx 180 ry 0 rz 180 deg; joints [-29.849, 20.571, 50.116, 60.045, 35.062, -54.852]
  Call Extruder(265.45163)
  MoveL 5270 to (237.3, 159.15, 78.65) mm, rotated rx 180 ry 0 rz 180 deg; joints [-29.907, 20.558, 50.134, 60.108, 35.106, -54.906]
  Call Extruder(266.27957)
  MoveL 5271 to (236.39, 160.19, 78.65) mm, rotated rx 180 ry 0 rz 180 deg; joints [-30.046, 20.499, 50.215, 60.274, 35.21, -55.052]
  Call Extruder(267.10752)
  MoveL 5272 to (235.35, 161.1, 78.65) mm, rotated rx 180 ry 0 rz 180 deg; joints [-30.182, 20.403, 50.345, 60.45, 35.304, -55.213]
  Call Extruder(267.27483)
  MoveL 5273 to (235.13, 161.27, 78.65) mm, rotated rx 180 ry 0 rz 180 deg; joints [-30.208, 20.379, 50.379, 60.487, 35.321, -55.248]
  MoveL 5274 to (235.13, 161.27, 78.65) mm, rotated rx 180 ry 0 rz 180 deg; joints [-30.208, 20.379, 50.379, 60.487, 35.321, -55.248]
  Call Extruder(267.60825)
  MoveL 5275 to (234.68, 161.6, 78.65) mm, rotated rx 180 ry 0 rz -180 deg; joints [-30.261, 20.33, 50.445, 60.561, 35.356, -55.317]
  MoveL 5276 to (234.68, 161.6, 78.65) mm, rotated rx 180 ry 0 rz -180 deg; joints [-30.261, 20.33, 50.445, 60.561, 35.356, -55.317]
  Call Extruder(267.94049)
  MoveL 5277 to (234.23, 161.92, 78.65) mm, rotated rx -180 ry 0 rz -180 deg; joints [-30.314, 20.281, 50.511, 60.634, 35.391, -55.385]
  MoveL 5278 to (234.23, 161.92, 78.65) mm, rotated rx -180 ry 0 rz -180 deg; joints [-30.314, 20.281, 50.511, 60.634, 35.391, -55.385]
  Call Extruder(268.05815)
  MoveL 5279 to (234.05, 162.02, 78.65) mm, rotated rx -180 ry 0 rz 180 deg; joints [-30.331, 20.26, 50.54, 60.661, 35.402, -55.411]
  MoveL 5280 to (234.05, 162.02, 78.65) mm, rotated rx -180 ry 0 rz 180 deg; joints [-30.331, 20.26, 50.54, 60.661, 35.402, -55.411]
  Call Extruder(268.26588)
  MoveL 5281 to (233.75, 162.2, 78.65) mm, rotated rx 180 ry 0 rz 180 deg; joints [-30.363, 20.223, 50.591, 60.708, 35.421, -55.456]
  MoveL 5282 to (233.75, 162.2, 78.65) mm, rotated rx 180 ry 0 rz 180 deg; joints [-30.363, 20.223, 50.591, 60.708, 35.421, -55.456]
  Call Extruder(268.47282)
  MoveL 5283 to (233.45, 162.37, 78.65) mm, rotated rx 180 ry 0 rz -180 deg; joints [-30.394, 20.185, 50.642, 60.755, 35.44, -55.502]
  MoveL 5284 to (233.45, 162.37, 78.65) mm, rotated rx 180 ry 0 rz -180 deg; joints [-30.394, 20.185, 50.642, 60.755, 35.44, -55.502]
  Call Extruder(268.67899)
  MoveL 5285 to (233.14, 162.55, 78.65) mm, rotated rx 180 ry 0 rz 180 deg; joints [-30.426, 20.147, 50.693, 60.803, 35.46, -55.547]
  MoveL 5286 to (233.14, 162.55, 78.65) mm, rotated rx 180 ry 0 rz 180 deg; joints [-30.426, 20.147, 50.693, 60.803, 35.46, -55.547]
  Call Extruder(268.86066)
  MoveL 5287 to (232.87, 162.69, 78.65) mm, rotated rx 180 ry 0 rz 180 deg; joints [-30.453, 20.111, 50.742, 60.845, 35.476, -55.588]
  MoveL 5288 to (232.87, 162.69, 78.65) mm, rotated rx 180 ry 0 rz 180 deg; joints [-30.453, 20.111, 50.742, 60.845, 35.476, -55.588]
  Call Extruder(269.01864)
  MoveL 5289 to (232.62, 162.8, 78.65) mm, rotated rx -180 ry 0 rz 180 deg; joints [-30.476, 20.077, 50.789, 60.882, 35.489, -55.624]
  MoveL 5290 to (232.62, 162.8, 78.65) mm, rotated rx -180 ry 0 rz 180 deg; joints [-30.476, 20.077, 50.789, 60.882, 35.489, -55.624]
  Call Extruder(269.17601)
  MoveL 5291 to (232.37, 162.9, 78.65) mm, rotated rx 180 ry 0 rz 180 deg; joints [-30.498, 20.042, 50.836, 60.919, 35.501, -55.661]
  MoveL 5292 to (232.37, 162.9, 78.65) mm, rotated rx 180 ry 0 rz 180 deg; joints [-30.498, 20.042, 50.836, 60.919, 35.501, -55.661]
  Call Extruder(269.35875)
  MoveL 5293 to (232.07, 163.02, 78.65) mm, rotated rx 180 ry 0 rz 180 deg; joints [-30.524, 20.001, 50.891, 60.962, 35.516, -55.703]
  MoveL 5294 to (232.07, 163.02, 78.65) mm, rotated rx 180 ry 0 rz 180 deg; joints [-30.524, 20.001, 50.891, 60.962, 35.516, -55.703]
  Call Extruder(269.54073)
  MoveL 5295 to (231.78, 163.15, 78.65) mm, rotated rx 180 ry 0 rz 180 deg; joints [-30.551, 19.96, 50.947, 61.005, 35.531, -55.745]
  MoveL 5296 to (231.78, 163.15, 78.65) mm, rotated rx 180 ry 0 rz 180 deg; joints [-30.551, 19.96, 50.947, 61.005, 35.531, -55.745]
  Call Extruder(269.68807)
  MoveL 5297 to (231.54, 163.24, 78.65) mm, rotated rx 180 ry 0 rz -180 deg; joints [-30.571, 19.926, 50.993, 61.04, 35.542, -55.78]
  MoveL 5298 to (231.54, 163.24, 78.65) mm, rotated rx 180 ry 0 rz -180 deg; joints [-30.571, 19.926, 50.993, 61.04, 35.542, -55.78]
  Call Extruder(269.80129)
  MoveL 5299 to (231.35, 163.3, 78.65) mm, rotated rx 180 ry 0 rz -180 deg; joints [-30.587, 19.897, 51.031, 61.067, 35.55, -55.807]
  MoveL 5300 to (231.35, 163.3, 78.65) mm, rotated rx 180 ry 0 rz -180 deg; joints [-30.587, 19.897, 51.031, 61.067, 35.55, -55.807]
  Call Extruder(269.91407)
  MoveL 5301 to (231.17, 163.36, 78.65) mm, rotated rx 180 ry 0 rz -180 deg; joints [-30.602, 19.869, 51.069, 61.094, 35.558, -55.834]
  MoveL 5302 to (231.17, 163.36, 78.65) mm, rotated rx 180 ry 0 rz -180 deg; joints [-30.602, 19.869, 51.069, 61.094, 35.558, -55.834]
  Call Extruder(270.02640)
  MoveL 5303 to (230.98, 163.42, 78.65) mm, rotated rx -180 ry 0 rz 180 deg; joints [-30.618, 19.841, 51.108, 61.121, 35.566, -55.861]
  MoveL 5304 to (230.98, 163.42, 78.65) mm, rotated rx -180 ry 0 rz 180 deg; joints [-30.618, 19.841, 51.108, 61.121, 35.566, -55.861]
  Call Extruder(270.13829)
  MoveL 5305 to (230.79, 163.48, 78.65) mm, rotated rx 180 ry 0 rz 180 deg; joints [-30.633, 19.813, 51.145, 61.148, 35.574, -55.888]
  MoveL 5306 to (230.79, 163.48, 78.65) mm, rotated rx 180 ry 0 rz 180 deg; joints [-30.633, 19.813, 51.145, 61.148, 35.574, -55.888]
  Call Extruder(270.25969)
  MoveL 5307 to (230.58, 163.55, 78.65) mm, rotated rx 180 ry 0 rz 180 deg; joints [-30.65, 19.782, 51.187, 61.177, 35.582, -55.917]
  MoveL 5308 to (230.58, 163.55, 78.65) mm, rotated rx 180 ry 0 rz 180 deg; joints [-30.65, 19.782, 51.187, 61.177, 35.582, -55.917]
  Call Extruder(270.39051)
  MoveL 5309 to (230.36, 163.61, 78.65) mm, rotated rx 180 ry 0 rz 180 deg; joints [-30.668, 19.748, 51.233, 61.209, 35.592, -55.949]
  MoveL 5310 to (230.36, 163.61, 78.65) mm, rotated rx 180 ry 0 rz 180 deg; joints [-30.668, 19.748, 51.233, 61.209, 35.592, -55.949]
  Call Extruder(270.52075)
  MoveL 5311 to (230.14, 163.68, 78.65) mm, rotated rx 180 ry 0 rz 180 deg; joints [-30.685, 19.715, 51.278, 61.24, 35.601, -55.981]
  MoveL 5312 to (230.14, 163.68, 78.65) mm, rotated rx 180 ry 0 rz 180 deg; joints [-30.685, 19.715, 51.278, 61.24, 35.601, -55.981]
  Call Extruder(270.65044)
  MoveL 5313 to (229.91, 163.75, 78.65) mm, rotated rx 180 ry 0 rz 180 deg; joints [-30.703, 19.681, 51.324, 61.272, 35.61, -56.012]
  MoveL 5314 to (229.91, 163.75, 78.65) mm, rotated rx 180 ry 0 rz 180 deg; joints [-30.703, 19.681, 51.324, 61.272, 35.61, -56.012]
  Call Extruder(270.77955)
  MoveL 5315 to (229.69, 163.82, 78.65) mm, rotated rx -180 ry 0 rz 180 deg; joints [-30.721, 19.647, 51.369, 61.304, 35.619, -56.044]
  MoveL 5316 to (229.69, 163.82, 78.65) mm, rotated rx -180 ry 0 rz 180 deg; joints [-30.721, 19.647, 51.369, 61.304, 35.619, -56.044]
  Call Extruder(270.89463)
  MoveL 5317 to (229.48, 163.86, 78.65) mm, rotated rx 180 ry 0 rz 180 deg; joints [-30.736, 19.615, 51.413, 61.332, 35.626, -56.073]
  MoveL 5318 to (229.48, 163.86, 78.65) mm, rotated rx 180 ry 0 rz 180 deg; joints [-30.736, 19.615, 51.413, 61.332, 35.626, -56.073]
  Call Extruder(271.00925)
  MoveL 5319 to (229.28, 163.91, 78.65) mm, rotated rx -180 ry 0 rz 180 deg; joints [-30.751, 19.582, 51.457, 61.36, 35.633, -56.101]
  MoveL 5320 to (229.28, 163.91, 78.65) mm, rotated rx -180 ry 0 rz 180 deg; joints [-30.751, 19.582, 51.457, 61.36, 35.633, -56.101]
  Call Extruder(271.12342)
  MoveL 5321 to (229.08, 163.95, 78.65) mm, rotated rx 180 ry 0 rz 180 deg; joints [-30.766, 19.55, 51.5, 61.388, 35.64, -56.13]
  MoveL 5322 to (229.08, 163.95, 78.65) mm, rotated rx 180 ry 0 rz 180 deg; joints [-30.766, 19.55, 51.5, 61.388, 35.64, -56.13]
  Call Extruder(271.23713)
  MoveL 5323 to (228.87, 164, 78.65) mm, rotated rx 180 ry 0 rz 180 deg; joints [-30.781, 19.517, 51.544, 61.416, 35.647, -56.158]
  MoveL 5324 to (228.87, 164, 78.65) mm, rotated rx 180 ry 0 rz 180 deg; joints [-30.781, 19.517, 51.544, 61.416, 35.647, -56.158]
  Call Extruder(271.36255)
  MoveL 5325 to (228.64, 164.04, 78.65) mm, rotated rx 180 ry 0 rz 180 deg; joints [-30.797, 19.481, 51.593, 61.446, 35.654, -56.189]
  MoveL 5326 to (228.64, 164.04, 78.65) mm, rotated rx 180 ry 0 rz 180 deg; joints [-30.797, 19.481, 51.593, 61.446, 35.654, -56.189]
  Call Extruder(271.49953)
  MoveL 5327 to (228.4, 164.09, 78.65) mm, rotated rx 180 ry 0 rz 180 deg; joints [-30.815, 19.441, 51.647, 61.48, 35.663, -56.224]
  MoveL 5328 to (228.4, 164.09, 78.65) mm, rotated rx 180 ry 0 rz 180 deg; joints [-30.815, 19.441, 51.647, 61.48, 35.663, -56.224]
  Call Extruder(271.63590)
  MoveL 5329 to (228.15, 164.14, 78.65) mm, rotated rx -180 ry 0 rz 180 deg; joints [-30.832, 19.401, 51.701, 61.514, 35.671, -56.258]
  MoveL 5330 to (228.15, 164.14, 78.65) mm, rotated rx -180 ry 0 rz 180 deg; joints [-30.832, 19.401, 51.701, 61.514, 35.671, -56.258]
  Call Extruder(271.77166)
  MoveL 5331 to (227.9, 164.19, 78.65) mm, rotated rx 180 ry 0 rz 180 deg; joints [-30.85, 19.361, 51.754, 61.547, 35.679, -56.293]
  MoveL 5332 to (227.9, 164.19, 78.65) mm, rotated rx 180 ry 0 rz 180 deg; joints [-30.85, 19.361, 51.754, 61.547, 35.679, -56.293]
  Call Extruder(271.90680)
  MoveL 5333 to (227.65, 164.24, 78.65) mm, rotated rx 180 ry 0 rz -180 deg; joints [-30.868, 19.321, 51.808, 61.581, 35.687, -56.327]
  MoveL 5334 to (227.65, 164.24, 78.65) mm, rotated rx 180 ry 0 rz -180 deg; joints [-30.868, 19.321, 51.808, 61.581, 35.687, -56.327]
  Call Extruder(272.04134)
  MoveL 5335 to (227.4, 164.29, 78.65) mm, rotated rx -180 ry 0 rz 180 deg; joints [-30.886, 19.281, 51.861, 61.614, 35.696, -56.361]
  MoveL 5336 to (227.4, 164.29, 78.65) mm, rotated rx -180 ry 0 rz 180 deg; joints [-30.886, 19.281, 51.861, 61.614, 35.696, -56.361]
  Call Extruder(272.17527)
  MoveL 5337 to (227.15, 164.34, 78.65) mm, rotated rx 180 ry 0 rz 180 deg; joints [-30.903, 19.241, 51.914, 61.648, 35.704, -56.395]
  MoveL 5338 to (227.15, 164.34, 78.65) mm, rotated rx 180 ry 0 rz 180 deg; joints [-30.903, 19.241, 51.914, 61.648, 35.704, -56.395]
  Call Extruder(272.32313)
  MoveL 5339 to (226.87, 164.39, 78.65) mm, rotated rx 180 ry 0 rz -180 deg; joints [-30.923, 19.196, 51.974, 61.685, 35.713, -56.433]
  MoveL 5340 to (226.87, 164.39, 78.65) mm, rotated rx 180 ry 0 rz -180 deg; joints [-30.923, 19.196, 51.974, 61.685, 35.713, -56.433]
  Call Extruder(272.48487)
  MoveL 5341 to (226.57, 164.44, 78.65) mm, rotated rx 180 ry 0 rz 180 deg; joints [-30.943, 19.146, 52.041, 61.725, 35.722, -56.474]
  MoveL 5342 to (226.57, 164.44, 78.65) mm, rotated rx 180 ry 0 rz 180 deg; joints [-30.943, 19.146, 52.041, 61.725, 35.722, -56.474]
  Call Extruder(272.64589)
  MoveL 5343 to (226.26, 164.49, 78.65) mm, rotated rx 180 ry 0 rz 180 deg; joints [-30.964, 19.096, 52.108, 61.765, 35.731, -56.516]
  MoveL 5344 to (226.26, 164.49, 78.65) mm, rotated rx 180 ry 0 rz 180 deg; joints [-30.964, 19.096, 52.108, 61.765, 35.731, -56.516]
  Call Extruder(272.80617)
  MoveL 5345 to (225.95, 164.53, 78.65) mm, rotated rx -180 ry 0 rz 180 deg; joints [-30.985, 19.046, 52.175, 61.806, 35.741, -56.557]
  MoveL 5346 to (225.95, 164.53, 78.65) mm, rotated rx -180 ry 0 rz 180 deg; joints [-30.985, 19.046, 52.175, 61.806, 35.741, -56.557]
  Call Extruder(272.96573)
  MoveL 5347 to (225.65, 164.58, 78.65) mm, rotated rx 180 ry 0 rz 180 deg; joints [-31.006, 18.997, 52.241, 61.846, 35.75, -56.598]
  MoveL 5348 to (225.65, 164.58, 78.65) mm, rotated rx 180 ry 0 rz 180 deg; joints [-31.006, 18.997, 52.241, 61.846, 35.75, -56.598]
  Call Extruder(273.12456)
  MoveL 5349 to (225.34, 164.63, 78.65) mm, rotated rx -180 ry 0 rz 180 deg; joints [-31.027, 18.947, 52.308, 61.886, 35.76, -56.639]
  MoveL 5350 to (225.34, 164.63, 78.65) mm, rotated rx -180 ry 0 rz 180 deg; joints [-31.027, 18.947, 52.308, 61.886, 35.76, -56.639]
  Call Extruder(273.30323)
  MoveL 5351 to (225, 164.68, 78.65) mm, rotated rx 180 ry 0 rz 180 deg; joints [-31.049, 18.89, 52.384, 61.931, 35.77, -56.685]
  MoveL 5352 to (225, 164.68, 78.65) mm, rotated rx 180 ry 0 rz 180 deg; joints [-31.049, 18.89, 52.384, 61.931, 35.77, -56.685]
  Call Extruder(273.50167)
  MoveL 5353 to (224.61, 164.72, 78.65) mm, rotated rx 180 ry 0 rz -180 deg; joints [-31.074, 18.825, 52.47, 61.98, 35.781, -56.737]
  MoveL 5354 to (224.61, 164.72, 78.65) mm, rotated rx 180 ry 0 rz -180 deg; joints [-31.074, 18.825, 52.47, 61.98, 35.781, -56.737]
  Call Extruder(273.69925)
  MoveL 5355 to (224.22, 164.77, 78.65) mm, rotated rx 180 ry 0 rz 180 deg; joints [-31.1, 18.761, 52.556, 62.03, 35.792, -56.788]
  MoveL 5356 to (224.22, 164.77, 78.65) mm, rotated rx 180 ry 0 rz 180 deg; joints [-31.1, 18.761, 52.556, 62.03, 35.792, -56.788]
  Call Extruder(273.89595)
  MoveL 5357 to (223.84, 164.82, 78.65) mm, rotated rx 180 ry 0 rz 180 deg; joints [-31.125, 18.697, 52.641, 62.079, 35.803, -56.839]
  MoveL 5358 to (223.84, 164.82, 78.65) mm, rotated rx 180 ry 0 rz 180 deg; joints [-31.125, 18.697, 52.641, 62.079, 35.803, -56.839]
  Call Extruder(274.09179)
  MoveL 5359 to (223.45, 164.86, 78.65) mm, rotated rx -180 ry 0 rz 180 deg; joints [-31.15, 18.632, 52.727, 62.129, 35.814, -56.89]
  MoveL 5360 to (223.45, 164.86, 78.65) mm, rotated rx -180 ry 0 rz 180 deg; joints [-31.15, 18.632, 52.727, 62.129, 35.814, -56.89]
  Call Extruder(274.38715)
  MoveL 5361 to (222.86, 164.91, 78.65) mm, rotated rx 180 ry 0 rz 180 deg; joints [-31.186, 18.533, 52.859, 62.202, 35.829, -56.967]
  MoveL 5362 to (222.86, 164.91, 78.65) mm, rotated rx 180 ry 0 rz 180 deg; joints [-31.186, 18.533, 52.859, 62.202, 35.829, -56.967]
  Call Extruder(274.68118)
  MoveL 5363 to (222.27, 164.95, 78.65) mm, rotated rx -180 ry 0 rz 180 deg; joints [-31.222, 18.433, 52.991, 62.276, 35.844, -57.043]
  MoveL 5364 to (222.27, 164.95, 78.65) mm, rotated rx -180 ry 0 rz 180 deg; joints [-31.222, 18.433, 52.991, 62.276, 35.844, -57.043]
  Call Extruder(274.97387)
  MoveL 5365 to (221.68, 165, 78.65) mm, rotated rx -180 ry 0 rz 180 deg; joints [-31.258, 18.334, 53.122, 62.349, 35.86, -57.119]
  MoveL 5366 to (221.68, 165, 78.65) mm, rotated rx -180 ry 0 rz 180 deg; joints [-31.258, 18.334, 53.122, 62.349, 35.86, -57.119]
  Call Extruder(275.54732)
  MoveL 5367 to (220.52, 165.05, 78.65) mm, rotated rx -180 ry 0 rz -180 deg; joints [-31.326, 18.134, 53.386, 62.49, 35.887, -57.267]
  MoveL 5368 to (220.52, 165.05, 78.65) mm, rotated rx -180 ry 0 rz -180 deg; joints [-31.326, 18.134, 53.386, 62.49, 35.887, -57.267]
  Call Extruder(276.26133)
  MoveL 5369 to (219.06, 165.09, 78.65) mm, rotated rx 180 ry 0 rz 180 deg; joints [-31.409, 17.884, 53.716, 62.664, 35.92, -57.449]
  Call Extruder(393.10807)
  MoveL 5370 to (-19.06, 165.09, 78.65) mm, rotated rx -180 ry 0 rz 180 deg; joints [-51.475, -11.844, 85.02, 77.023, 53.402, -68.868]
  Call Extruder(393.53667)
  MoveL 5371 to (-19.94, 165.07, 78.65) mm, rotated rx -180 ry 0 rz 180 deg; joints [-51.582, -11.924, 85.083, 77.059, 53.506, -68.876]
  MoveL 5372 to (-19.94, 165.07, 78.65) mm, rotated rx -180 ry 0 rz 180 deg; joints [-51.582, -11.924, 85.083, 77.059, 53.506, -68.876]
  Call Extruder(394.11012)
  MoveL 5373 to (-21.1, 165.03, 78.65) mm, rotated rx -180 ry 0 rz -180 deg; joints [-51.722, -12.033, 85.169, 77.106, 53.642, -68.886]
  MoveL 5374 to (-21.1, 165.03, 78.65) mm, rotated rx -180 ry 0 rz -180 deg; joints [-51.722, -12.033, 85.169, 77.106, 53.642, -68.886]
  Call Extruder(394.54442)
  MoveL 5375 to (-21.97, 164.98, 78.65) mm, rotated rx 180 ry 0 rz 180 deg; joints [-51.827, -12.115, 85.234, 77.14, 53.743, -68.892]
  MoveL 5376 to (-21.97, 164.98, 78.65) mm, rotated rx 180 ry 0 rz 180 deg; joints [-51.827, -12.115, 85.234, 77.14, 53.743, -68.892]
  Call Extruder(394.83845)
  MoveL 5377 to (-22.56, 164.93, 78.65) mm, rotated rx 180 ry 0 rz -180 deg; joints [-51.897, -12.173, 85.279, 77.162, 53.811, -68.896]
  MoveL 5378 to (-22.56, 164.93, 78.65) mm, rotated rx 180 ry 0 rz -180 deg; joints [-51.897, -12.173, 85.279, 77.162, 53.811, -68.896]
  Call Extruder(395.13381)
  MoveL 5379 to (-23.15, 164.89, 78.65) mm, rotated rx 180 ry 0 rz 180 deg; joints [-51.966, -12.23, 85.324, 77.185, 53.878, -68.899]
  MoveL 5380 to (-23.15, 164.89, 78.65) mm, rotated rx 180 ry 0 rz 180 deg; joints [-51.966, -12.23, 85.324, 77.185, 53.878, -68.899]
  Call Extruder(395.38003)
  MoveL 5381 to (-23.64, 164.84, 78.65) mm, rotated rx 180 ry 0 rz 180 deg; joints [-52.023, -12.278, 85.362, 77.203, 53.934, -68.902]
  MoveL 5382 to (-23.64, 164.84, 78.65) mm, rotated rx 180 ry 0 rz 180 deg; joints [-52.023, -12.278, 85.362, 77.203, 53.934, -68.902]
  Call Extruder(395.57673)
  MoveL 5383 to (-24.03, 164.79, 78.65) mm, rotated rx 180 ry 0 rz 180 deg; joints [-52.067, -12.318, 85.393, 77.216, 53.977, -68.903]
  MoveL 5384 to (-24.03, 164.79, 78.65) mm, rotated rx 180 ry 0 rz 180 deg; joints [-52.067, -12.318, 85.393, 77.216, 53.977, -68.903]
  Call Extruder(395.77431)
  MoveL 5385 to (-24.42, 164.75, 78.65) mm, rotated rx -180 ry 0 rz 180 deg; joints [-52.112, -12.357, 85.424, 77.23, 54.02, -68.905]
  MoveL 5386 to (-24.42, 164.75, 78.65) mm, rotated rx -180 ry 0 rz 180 deg; joints [-52.112, -12.357, 85.424, 77.23, 54.02, -68.905]
  Call Extruder(395.97275)
  MoveL 5387 to (-24.8, 164.7, 78.65) mm, rotated rx 180 ry 0 rz 180 deg; joints [-52.156, -12.396, 85.454, 77.244, 54.064, -68.906]
  MoveL 5388 to (-24.8, 164.7, 78.65) mm, rotated rx 180 ry 0 rz 180 deg; joints [-52.156, -12.396, 85.454, 77.244, 54.064, -68.906]
  Call Extruder(396.17206)
  MoveL 5389 to (-25.19, 164.66, 78.65) mm, rotated rx 180 ry 0 rz -180 deg; joints [-52.2, -12.435, 85.485, 77.258, 54.107, -68.907]
  MoveL 5390 to (-25.19, 164.66, 78.65) mm, rotated rx 180 ry 0 rz -180 deg; joints [-52.2, -12.435, 85.485, 77.258, 54.107, -68.907]
  Call Extruder(396.33089)
  MoveL 5391 to (-25.5, 164.61, 78.65) mm, rotated rx 180 ry 0 rz 180 deg; joints [-52.235, -12.467, 85.51, 77.268, 54.14, -68.908]
  MoveL 5392 to (-25.5, 164.61, 78.65) mm, rotated rx 180 ry 0 rz 180 deg; joints [-52.235, -12.467, 85.51, 77.268, 54.14, -68.908]
  Call Extruder(396.49045)
  MoveL 5393 to (-25.8, 164.56, 78.65) mm, rotated rx -180 ry 0 rz -180 deg; joints [-52.269, -12.5, 85.535, 77.278, 54.173, -68.908]
  MoveL 5394 to (-25.8, 164.56, 78.65) mm, rotated rx -180 ry 0 rz -180 deg; joints [-52.269, -12.5, 85.535, 77.278, 54.173, -68.908]
  Call Extruder(396.65073)
  MoveL 5395 to (-26.11, 164.51, 78.65) mm, rotated rx 180 ry 0 rz -180 deg; joints [-52.303, -12.532, 85.561, 77.288, 54.207, -68.909]
  MoveL 5396 to (-26.11, 164.51, 78.65) mm, rotated rx 180 ry 0 rz -180 deg; joints [-52.303, -12.532, 85.561, 77.288, 54.207, -68.909]
  Call Extruder(396.81175)
  MoveL 5397 to (-26.41, 164.46, 78.65) mm, rotated rx 180 ry 0 rz 180 deg; joints [-52.337, -12.564, 85.586, 77.298, 54.24, -68.909]
  MoveL 5398 to (-26.41, 164.46, 78.65) mm, rotated rx 180 ry 0 rz 180 deg; joints [-52.337, -12.564, 85.586, 77.298, 54.24, -68.909]
  Call Extruder(396.97349)
  MoveL 5399 to (-26.72, 164.41, 78.65) mm, rotated rx -180 ry 0 rz 180 deg; joints [-52.371, -12.596, 85.611, 77.308, 54.274, -68.909]
  MoveL 5400 to (-26.72, 164.41, 78.65) mm, rotated rx -180 ry 0 rz 180 deg; joints [-52.371, -12.596, 85.611, 77.308, 54.274, -68.909]
  Call Extruder(397.13596)
  MoveL 5401 to (-27.02, 164.37, 78.65) mm, rotated rx 180 ry 0 rz -180 deg; joints [-52.405, -12.628, 85.636, 77.319, 54.307, -68.91]
  MoveL 5402 to (-27.02, 164.37, 78.65) mm, rotated rx 180 ry 0 rz -180 deg; joints [-52.405, -12.628, 85.636, 77.319, 54.307, -68.91]
  Call Extruder(397.26988)
  MoveL 5403 to (-27.27, 164.32, 78.65) mm, rotated rx 180 ry 0 rz 180 deg; joints [-52.432, -12.656, 85.657, 77.326, 54.333, -68.909]
  MoveL 5404 to (-27.27, 164.32, 78.65) mm, rotated rx 180 ry 0 rz 180 deg; joints [-52.432, -12.656, 85.657, 77.326, 54.333, -68.909]
  Call Extruder(397.40442)
  MoveL 5405 to (-27.52, 164.27, 78.65) mm, rotated rx 180 ry 0 rz 180 deg; joints [-52.459, -12.683, 85.678, 77.334, 54.36, -68.909]
  MoveL 5406 to (-27.52, 164.27, 78.65) mm, rotated rx 180 ry 0 rz 180 deg; joints [-52.459, -12.683, 85.678, 77.334, 54.36, -68.909]
  Call Extruder(397.53957)
  MoveL 5407 to (-27.77, 164.22, 78.65) mm, rotated rx 180 ry 0 rz 180 deg; joints [-52.486, -12.71, 85.7, 77.342, 54.386, -68.909]
  MoveL 5408 to (-27.77, 164.22, 78.65) mm, rotated rx 180 ry 0 rz 180 deg; joints [-52.486, -12.71, 85.7, 77.342, 54.386, -68.909]
  Call Extruder(397.67532)
  MoveL 5409 to (-28.02, 164.17, 78.65) mm, rotated rx 180 ry 0 rz -180 deg; joints [-52.513, -12.737, 85.721, 77.349, 54.413, -68.908]
  MoveL 5410 to (-28.02, 164.17, 78.65) mm, rotated rx 180 ry 0 rz -180 deg; joints [-52.513, -12.737, 85.721, 77.349, 54.413, -68.908]
  Call Extruder(397.81169)
  MoveL 5411 to (-28.27, 164.12, 78.65) mm, rotated rx 180 ry 0 rz 180 deg; joints [-52.54, -12.765, 85.742, 77.357, 54.439, -68.908]
  MoveL 5412 to (-28.27, 164.12, 78.65) mm, rotated rx 180 ry 0 rz 180 deg; joints [-52.54, -12.765, 85.742, 77.357, 54.439, -68.908]
  Call Extruder(397.89656)
  MoveL 5413 to (-28.43, 164.09, 78.65) mm, rotated rx 180 ry 0 rz 180 deg; joints [-52.556, -12.781, 85.755, 77.362, 54.456, -68.908]
  Set speed (130.0 mm/s)
  MoveL 5414 to (-31.76, 163.31, 78.65) mm, rotated rx -180 ry 0 rz 180 deg; joints [-52.91, -13.157, 86.045, 77.459, 54.804, -68.896]
  MoveL 5415 to (-31.76, 163.31, 88.06) mm, rotated rx 180 ry 0 rz 180 deg; joints [-52.91, -13.899, 88.098, 78.367, 54.529, -70.466]
  Call Extruder(395.89656)
  Set speed (40.0 mm/s)
  MoveL 5416 to (-31.76, 163.31, 88.06) mm, rotated rx 180 ry 0 rz 180 deg; joints [-52.91, -13.899, 88.098, 78.367, 54.529, -70.466]
  Call Extruder(0.00000)
  Set speed (130.0 mm/s)
  MoveL 5417 to (-31.64, 163.21, 88.06) mm, rotated rx 180 ry 0 rz 180 deg; joints [-52.884, -13.901, 88.099, 78.356, 54.505, -70.46]
  Call Extruder(2.00000)
  Set speed (40.0 mm/s)
  MoveL 5418 to (-31.64, 163.21, 88.06) mm, rotated rx 180 ry 0 rz 180 deg; joints [-52.884, -13.901, 88.099, 78.356, 54.505, -70.46]
  Set speed (30.0 mm/s)
